// TIA Portal V15.1 export
// export: Created 2024-05-17T05:38:30.0630205Z, ExportSetting WithDefaults, DisplayName Totally Integrated Automation Portal, DisplayVersion V15.1 Update 5, DisplayName TIA Portal Openness, DisplayVersion V15.1 Update 5, DisplayName SINAMICS Startdrive Advanced, DisplayVersion V15.1, DisplayName G130, G150, S120, S150, SINAMICS MV, S210, DisplayVersion V15.1, DisplayName G110M, G120, G120C, G120D, G120P, DisplayVersion V15.1, DisplayName STEP 7 Professional, DisplayVersion V15.1 Update 5, DisplayName STEP 7 Safety, DisplayVersion V15.1, DisplayName WinCC Professional, DisplayVersion V15.1 Update 5, DisplayName SIMATIC Visualization Architect, DisplayVersion V15.1
FUNCTION_BLOCK "LComAlarm"   // FB2105, FBD
TITLE = LComAlarm
{ S7_Optimized_Access := 'FALSE' }
AUTHOR : VCC
FAMILY : Communic
VERSION : 0.1
// =============================================================================
// This module Handles All Alarm Report To MES/VD
// =============================================================================
// stored: AutoNumber false, IsIECCheckEnabled false, SetENOAutomatically False, UDAEnableTagReadback false
   VAR_INPUT
      C_VDCommRecvDB { ExternalAccessible := 'False'; ExternalVisible := 'False'; ExternalWritable := 'False'} : DB_ANY;   // VD communication system receive DB; Not to be used by application / VD communication system receive DB; Not to be used by Application
      C_VDCommSendDB { ExternalAccessible := 'False'; ExternalVisible := 'False'; ExternalWritable := 'False'} : DB_ANY;   // VD communication system send DB; Not to be used by application / VD communication system send DB; Not to be used by Application
      C_LocalRecvDB { ExternalAccessible := 'False'; ExternalVisible := 'False'; ExternalWritable := 'False'} : DB_ANY;   // Local DB to store received data; to used by application / Local DB For Recv Data Used By The Application
      C_LocalSendDB { ExternalAccessible := 'False'; ExternalVisible := 'False'; ExternalWritable := 'False'} : DB_ANY;   // Local DB for send data; to be used by application / Local DB For Send Data Used By The Application
      C_GenAlarmDB { ExternalAccessible := 'False'; ExternalVisible := 'False'; ExternalWritable := 'False'} : DB_ANY;   // Alarm DB
      C_AlarmDBMZ1 { ExternalAccessible := 'False'; ExternalVisible := 'False'; ExternalWritable := 'False'} : DB_ANY;   // Alarm DB
      C_AlarmDBMZ2 { ExternalAccessible := 'False'; ExternalVisible := 'False'; ExternalWritable := 'False'} : DB_ANY;   // Alarm DB
      C_AlarmDBMZ3 { ExternalAccessible := 'False'; ExternalVisible := 'False'; ExternalWritable := 'False'} : DB_ANY;   // Alarm DB
      C_AlarmDBMZ4 { ExternalAccessible := 'False'; ExternalVisible := 'False'; ExternalWritable := 'False'} : DB_ANY;   // Alarm DB
      C_AlarmDBMZ5 { ExternalAccessible := 'False'; ExternalVisible := 'False'; ExternalWritable := 'False'} : DB_ANY;   // Alarm DB
      C_AlarmDBMZ6 { ExternalAccessible := 'False'; ExternalVisible := 'False'; ExternalWritable := 'False'} : DB_ANY;   // Alarm DB
      C_AlarmDBMZ7 { ExternalAccessible := 'False'; ExternalVisible := 'False'; ExternalWritable := 'False'} : DB_ANY;   // Alarm DB
      C_AlarmDBMZ8 { ExternalAccessible := 'False'; ExternalVisible := 'False'; ExternalWritable := 'False'} : DB_ANY;   // Alarm DB
      C_AlarmDBMZ9 { ExternalAccessible := 'False'; ExternalVisible := 'False'; ExternalWritable := 'False'} : DB_ANY;   // Alarm DB
      C_AlarmDBMZ10 { ExternalAccessible := 'False'; ExternalVisible := 'False'; ExternalWritable := 'False'} : DB_ANY;   // Alarm DB
      C_AlarmDBMZ11 { ExternalAccessible := 'False'; ExternalVisible := 'False'; ExternalWritable := 'False'} : DB_ANY;   // Alarm DB
      C_AlarmDBMZ12 { ExternalAccessible := 'False'; ExternalVisible := 'False'; ExternalWritable := 'False'} : DB_ANY;   // Alarm DB
      C_AlarmDBMZ13 { ExternalAccessible := 'False'; ExternalVisible := 'False'; ExternalWritable := 'False'} : DB_ANY;   // Alarm DB
      C_AlarmDBMZ14 { ExternalAccessible := 'False'; ExternalVisible := 'False'; ExternalWritable := 'False'} : DB_ANY;   // Alarm DB
      C_GenAlarmCompare { ExternalAccessible := 'False'; ExternalVisible := 'False'; ExternalWritable := 'False'} : DB_ANY;   // Alarm DB
      C_AlarmCompareDBMZ1 { ExternalAccessible := 'False'; ExternalVisible := 'False'; ExternalWritable := 'False'} : DB_ANY;   // Alarm DB
      C_AlarmCompareDBMZ2 { ExternalAccessible := 'False'; ExternalVisible := 'False'; ExternalWritable := 'False'} : DB_ANY;   // Alarm DB
      C_AlarmCompareDBMZ3 { ExternalAccessible := 'False'; ExternalVisible := 'False'; ExternalWritable := 'False'} : DB_ANY;   // Alarm DB
      C_AlarmCompareDBMZ4 { ExternalAccessible := 'False'; ExternalVisible := 'False'; ExternalWritable := 'False'} : DB_ANY;   // Alarm DB
      C_AlarmCompareDBMZ5 { ExternalAccessible := 'False'; ExternalVisible := 'False'; ExternalWritable := 'False'} : DB_ANY;   // Alarm DB
      C_AlarmCompareDBMZ6 { ExternalAccessible := 'False'; ExternalVisible := 'False'; ExternalWritable := 'False'} : DB_ANY;   // Alarm DB
      C_AlarmCompareDBMZ7 { ExternalAccessible := 'False'; ExternalVisible := 'False'; ExternalWritable := 'False'} : DB_ANY;   // Alarm DB
      C_AlarmCompareDBMZ8 { ExternalAccessible := 'False'; ExternalVisible := 'False'; ExternalWritable := 'False'} : DB_ANY;   // Alarm DB
      C_AlarmCompareDBMZ9 { ExternalAccessible := 'False'; ExternalVisible := 'False'; ExternalWritable := 'False'} : DB_ANY;   // Alarm DB
      C_AlarmCompareDBMZ10 { ExternalAccessible := 'False'; ExternalVisible := 'False'; ExternalWritable := 'False'} : DB_ANY;   // Alarm DB
      C_AlarmCompareDBMZ11 { ExternalAccessible := 'False'; ExternalVisible := 'False'; ExternalWritable := 'False'} : DB_ANY;   // Alarm DB
      C_AlarmCompareDBMZ12 { ExternalAccessible := 'False'; ExternalVisible := 'False'; ExternalWritable := 'False'} : DB_ANY;   // Alarm DB
      C_AlarmCompareDBMZ13 { ExternalAccessible := 'False'; ExternalVisible := 'False'; ExternalWritable := 'False'} : DB_ANY;   // Alarm DB
      C_AlarmCompareDBMZ14 { ExternalAccessible := 'False'; ExternalVisible := 'False'; ExternalWritable := 'False'} : DB_ANY;   // Alarm DB
      C_SubSystem { ExternalAccessible := 'False'; ExternalVisible := 'False'; ExternalWritable := 'False'} : Int;   // Number to identify the subsystem / Identify Subsystem
      C_SendDelay { ExternalAccessible := 'False'; ExternalVisible := 'False'; ExternalWritable := 'False'} : DInt;   // Send Alarm Delay
      C_NbrOfModeZone { ExternalAccessible := 'False'; ExternalVisible := 'False'; ExternalWritable := 'False'} : Int;   // Nbr Of ModeZones
      C_Filter { ExternalAccessible := 'False'; ExternalVisible := 'False'; ExternalWritable := 'False'} : Time := T#500ms;   // Filter
   END_VAR
   VAR_IN_OUT
      IO_VD : "VDComm";   // VD Comm
      IO_AlarmDB : "AlarmDB";   // Alarm
   END_VAR
   VAR
      _LVDComSubSystem { ExternalAccessible := 'False'; ExternalVisible := 'False'; ExternalWritable := 'False'; S7_SetPoint := 'True'} : "LVDComSubSystemS7-1500";   // VD Sub System Alarm
   END_VAR
   VAR DB_SPECIFIC
      ReqSendToVDAlarm { ExternalAccessible := 'False'; ExternalVisible := 'False'; ExternalWritable := 'False'} : Array[1..32] of Bool;   // Req VD
      SendAlarm { ExternalAccessible := 'False'; ExternalVisible := 'False'; ExternalWritable := 'False'} : Array[1..64] of Bool;   // Req Send Alarm
      SendAlarmDone { ExternalAccessible := 'False'; ExternalVisible := 'False'; ExternalWritable := 'False'} : Array[1..64] of Bool;   // Change Of State
      ActiveRequest { ExternalAccessible := 'False'; ExternalVisible := 'False'; ExternalWritable := 'False'} : DWord;   // No Requests Active
      OkToRequest { ExternalAccessible := 'False'; ExternalVisible := 'False'; ExternalWritable := 'False'} : Bool;   // Ok To Request New Alarm To VD
      SendDoneVD { ExternalAccessible := 'False'; ExternalVisible := 'False'; ExternalWritable := 'False'} : Bool;   // Request Is Finished
      SendToVD { ExternalAccessible := 'False'; ExternalVisible := 'False'; ExternalWritable := 'False'} : Bool;   // Send To VD
      InitUDT { ExternalAccessible := 'False'; ExternalVisible := 'False'; ExternalWritable := 'False'} : Bool;   // Init
      DelaySend { ExternalAccessible := 'False'; ExternalVisible := 'False'; ExternalWritable := 'False'} : Bool;   // Delay Send To VD
      InitSend { ExternalAccessible := 'False'; ExternalVisible := 'False'; ExternalWritable := 'False'} : Bool;   // Init Send
      ResetSendDone { ExternalAccessible := 'False'; ExternalVisible := 'False'; ExternalWritable := 'False'} : Bool;   // Reset Send Done
      ResetAllRequest { ExternalAccessible := 'False'; ExternalVisible := 'False'; ExternalWritable := 'False'} : Bool;   // Reset All Send Requests
      Edge { ExternalAccessible := 'False'; ExternalVisible := 'False'; ExternalWritable := 'False'} : Array[1..64] of Bool;   // Array
      SendDBNbr { ExternalAccessible := 'False'; ExternalVisible := 'False'; ExternalWritable := 'False'} : Int;   // Pointer
      SendDBBufNbr { ExternalAccessible := 'False'; ExternalVisible := 'False'; ExternalWritable := 'False'} : Int;   // Pointer
      AlarmPointer { ExternalAccessible := 'False'; ExternalVisible := 'False'; ExternalWritable := 'False'} : Word;   // Pointer
      AlarmLength { ExternalAccessible := 'False'; ExternalVisible := 'False'; ExternalWritable := 'False'} : Word;   // Pointer
      SendLength { ExternalAccessible := 'False'; ExternalVisible := 'False'; ExternalWritable := 'False'} : Word;   // Pointer
      SendDoneArr { ExternalAccessible := 'False'; ExternalVisible := 'False'; ExternalWritable := 'False'} : Array[0..1] of DWord;   // Array Send Done
   END_VAR
   VAR
      _DelaySend { ExternalAccessible := 'False'; ExternalVisible := 'False'; ExternalWritable := 'False'; S7_SetPoint := 'True'} : "LTimer";   // FB
      _LMDBToDBGen { ExternalAccessible := 'False'; ExternalVisible := 'False'; ExternalWritable := 'False'; S7_SetPoint := 'True'} : "LMDBToDB";   // FB
      _LMDBToDBMZ1 { ExternalAccessible := 'False'; ExternalVisible := 'False'; ExternalWritable := 'False'; S7_SetPoint := 'True'} : "LMDBToDB";   // FB
      _LMDBToDBMZ2 { ExternalAccessible := 'False'; ExternalVisible := 'False'; ExternalWritable := 'False'; S7_SetPoint := 'True'} : "LMDBToDB";   // FB
      _LMDBToDBMZ3 { ExternalAccessible := 'False'; ExternalVisible := 'False'; ExternalWritable := 'False'; S7_SetPoint := 'True'} : "LMDBToDB";   // FB
      _LMDBToDBMZ4 { ExternalAccessible := 'False'; ExternalVisible := 'False'; ExternalWritable := 'False'; S7_SetPoint := 'True'} : "LMDBToDB";   // FB
      _LMDBToDBMZ5 { ExternalAccessible := 'False'; ExternalVisible := 'False'; ExternalWritable := 'False'; S7_SetPoint := 'True'} : "LMDBToDB";   // FB
      _LMDBToDBMZ6 { ExternalAccessible := 'False'; ExternalVisible := 'False'; ExternalWritable := 'False'; S7_SetPoint := 'True'} : "LMDBToDB";   // FB
      _LMDBToDBMZ7 { ExternalAccessible := 'False'; ExternalVisible := 'False'; ExternalWritable := 'False'; S7_SetPoint := 'True'} : "LMDBToDB";   // FB
      _LMDBToDBMZ8 { ExternalAccessible := 'False'; ExternalVisible := 'False'; ExternalWritable := 'False'; S7_SetPoint := 'True'} : "LMDBToDB";   // FB
      _LMDBToDBMZ9 { ExternalAccessible := 'False'; ExternalVisible := 'False'; ExternalWritable := 'False'; S7_SetPoint := 'True'} : "LMDBToDB";   // FB
      _LMDBToDBMZ10 { ExternalAccessible := 'False'; ExternalVisible := 'False'; ExternalWritable := 'False'; S7_SetPoint := 'True'} : "LMDBToDB";   // FB
      _LMDBToDBMZ11 { ExternalAccessible := 'False'; ExternalVisible := 'False'; ExternalWritable := 'False'; S7_SetPoint := 'True'} : "LMDBToDB";   // FB
      _LMDBToDBMZ12 { ExternalAccessible := 'False'; ExternalVisible := 'False'; ExternalWritable := 'False'; S7_SetPoint := 'True'} : "LMDBToDB";   // FB
      _LMDBToDBMZ13 { ExternalAccessible := 'False'; ExternalVisible := 'False'; ExternalWritable := 'False'; S7_SetPoint := 'True'} : "LMDBToDB";   // FB
      _LMDBToDBMZ14 { ExternalAccessible := 'False'; ExternalVisible := 'False'; ExternalWritable := 'False'; S7_SetPoint := 'True'} : "LMDBToDB";   // FB
      _LDBCheckGen { ExternalAccessible := 'False'; ExternalVisible := 'False'; ExternalWritable := 'False'; S7_SetPoint := 'True'} : "LDBCheck";   // FB
      _LDBCheckMZ1 { ExternalAccessible := 'False'; ExternalVisible := 'False'; ExternalWritable := 'False'; S7_SetPoint := 'True'} : "LDBCheck";   // FB
      _LDBCheckMZ2 { ExternalAccessible := 'False'; ExternalVisible := 'False'; ExternalWritable := 'False'; S7_SetPoint := 'True'} : "LDBCheck";   // FB
      _LDBCheckMZ3 { ExternalAccessible := 'False'; ExternalVisible := 'False'; ExternalWritable := 'False'; S7_SetPoint := 'True'} : "LDBCheck";   // FB
      _LDBCheckMZ4 { ExternalAccessible := 'False'; ExternalVisible := 'False'; ExternalWritable := 'False'; S7_SetPoint := 'True'} : "LDBCheck";   // FB
      _LDBCheckMZ5 { ExternalAccessible := 'False'; ExternalVisible := 'False'; ExternalWritable := 'False'; S7_SetPoint := 'True'} : "LDBCheck";   // FB
      _LDBCheckMZ6 { ExternalAccessible := 'False'; ExternalVisible := 'False'; ExternalWritable := 'False'; S7_SetPoint := 'True'} : "LDBCheck";   // FB
      _LDBCheckMZ7 { ExternalAccessible := 'False'; ExternalVisible := 'False'; ExternalWritable := 'False'; S7_SetPoint := 'True'} : "LDBCheck";   // FB
      _LDBCheckMZ8 { ExternalAccessible := 'False'; ExternalVisible := 'False'; ExternalWritable := 'False'; S7_SetPoint := 'True'} : "LDBCheck";   // FB
      _LDBCheckMZ9 { ExternalAccessible := 'False'; ExternalVisible := 'False'; ExternalWritable := 'False'; S7_SetPoint := 'True'} : "LDBCheck";   // FB
      _LDBCheckMZ10 { ExternalAccessible := 'False'; ExternalVisible := 'False'; ExternalWritable := 'False'; S7_SetPoint := 'True'} : "LDBCheck";   // FB
      _LDBCheckMZ11 { ExternalAccessible := 'False'; ExternalVisible := 'False'; ExternalWritable := 'False'; S7_SetPoint := 'True'} : "LDBCheck";   // FB
      _LDBCheckMZ12 { ExternalAccessible := 'False'; ExternalVisible := 'False'; ExternalWritable := 'False'; S7_SetPoint := 'True'} : "LDBCheck";   // FB
      _LDBCheckMZ13 { ExternalAccessible := 'False'; ExternalVisible := 'False'; ExternalWritable := 'False'; S7_SetPoint := 'True'} : "LDBCheck";   // FB
      _LDBCheckMZ14 { ExternalAccessible := 'False'; ExternalVisible := 'False'; ExternalWritable := 'False'; S7_SetPoint := 'True'} : "LDBCheck";   // FB
   END_VAR
   VAR DB_SPECIFIC
      _SendDoneReset { ExternalAccessible := 'False'; ExternalVisible := 'False'; ExternalWritable := 'False'; S7_SetPoint := 'True'} : TON_TIME;   // FB
      Filter { ExternalAccessible := 'False'; ExternalVisible := 'False'; ExternalWritable := 'False'} : Array[1..16] of Bool;   // Array
      _FilterGen { ExternalAccessible := 'False'; ExternalVisible := 'False'; ExternalWritable := 'False'; S7_SetPoint := 'True'} : TON_TIME;   // FB
      _FilterMZ1 { ExternalAccessible := 'False'; ExternalVisible := 'False'; ExternalWritable := 'False'; S7_SetPoint := 'True'} : TON_TIME;   // FB
      _FilterMZ2 { ExternalAccessible := 'False'; ExternalVisible := 'False'; ExternalWritable := 'False'; S7_SetPoint := 'True'} : TON_TIME;   // FB
      _FilterMZ3 { ExternalAccessible := 'False'; ExternalVisible := 'False'; ExternalWritable := 'False'; S7_SetPoint := 'True'} : TON_TIME;   // FB
      _FilterMZ4 { ExternalAccessible := 'False'; ExternalVisible := 'False'; ExternalWritable := 'False'; S7_SetPoint := 'True'} : TON_TIME;   // FB
      _FilterMZ5 { ExternalAccessible := 'False'; ExternalVisible := 'False'; ExternalWritable := 'False'; S7_SetPoint := 'True'} : TON_TIME;   // FB
      _FilterMZ6 { ExternalAccessible := 'False'; ExternalVisible := 'False'; ExternalWritable := 'False'; S7_SetPoint := 'True'} : TON_TIME;   // FB
      _FilterMZ7 { ExternalAccessible := 'False'; ExternalVisible := 'False'; ExternalWritable := 'False'; S7_SetPoint := 'True'} : TON_TIME;   // FB
      _FilterMZ8 { ExternalAccessible := 'False'; ExternalVisible := 'False'; ExternalWritable := 'False'; S7_SetPoint := 'True'} : TON_TIME;   // FB
      _FilterMZ9 { ExternalAccessible := 'False'; ExternalVisible := 'False'; ExternalWritable := 'False'; S7_SetPoint := 'True'} : TON_TIME;   // FB
      _FilterMZ10 { ExternalAccessible := 'False'; ExternalVisible := 'False'; ExternalWritable := 'False'; S7_SetPoint := 'True'} : TON_TIME;   // FB
      _FilterMZ11 { ExternalAccessible := 'False'; ExternalVisible := 'False'; ExternalWritable := 'False'; S7_SetPoint := 'True'} : TON_TIME;   // FB
      _FilterMZ12 { ExternalAccessible := 'False'; ExternalVisible := 'False'; ExternalWritable := 'False'; S7_SetPoint := 'True'} : TON_TIME;   // FB
      _FilterMZ13 { ExternalAccessible := 'False'; ExternalVisible := 'False'; ExternalWritable := 'False'; S7_SetPoint := 'True'} : TON_TIME;   // FB
      _FilterMZ14 { ExternalAccessible := 'False'; ExternalVisible := 'False'; ExternalWritable := 'False'; S7_SetPoint := 'True'} : TON_TIME;   // FB
      _InitSend { ExternalAccessible := 'False'; ExternalVisible := 'False'; ExternalWritable := 'False'; S7_SetPoint := 'True'} : TON_TIME;   // FB
      GenDBLenghtOk { ExternalAccessible := 'False'; ExternalVisible := 'False'; ExternalWritable := 'False'} : Bool;   // DB Length Ok
      MZ1DBLenghtOk { ExternalAccessible := 'False'; ExternalVisible := 'False'; ExternalWritable := 'False'} : Bool;   // DB Length Ok
      MZ2DBLenghtOk { ExternalAccessible := 'False'; ExternalVisible := 'False'; ExternalWritable := 'False'} : Bool;   // DB Length Ok
      MZ3DBLenghtOk { ExternalAccessible := 'False'; ExternalVisible := 'False'; ExternalWritable := 'False'} : Bool;   // DB Length Ok
      MZ4DBLenghtOk { ExternalAccessible := 'False'; ExternalVisible := 'False'; ExternalWritable := 'False'} : Bool;   // DB Length Ok
      MZ5DBLenghtOk { ExternalAccessible := 'False'; ExternalVisible := 'False'; ExternalWritable := 'False'} : Bool;   // DB Length Ok
      MZ6DBLenghtOk { ExternalAccessible := 'False'; ExternalVisible := 'False'; ExternalWritable := 'False'} : Bool;   // DB Length Ok
      MZ7DBLenghtOk { ExternalAccessible := 'False'; ExternalVisible := 'False'; ExternalWritable := 'False'} : Bool;   // DB Length Ok
      MZ8DBLenghtOk { ExternalAccessible := 'False'; ExternalVisible := 'False'; ExternalWritable := 'False'} : Bool;   // DB Length Ok
      MZ9DBLenghtOk { ExternalAccessible := 'False'; ExternalVisible := 'False'; ExternalWritable := 'False'} : Bool;   // DB Length Ok
      MZ10DBLenghtOk { ExternalAccessible := 'False'; ExternalVisible := 'False'; ExternalWritable := 'False'} : Bool;   // DB Length Ok
      MZ11DBLenghtOk { ExternalAccessible := 'False'; ExternalVisible := 'False'; ExternalWritable := 'False'} : Bool;   // DB Length Ok
      MZ12DBLenghtOk { ExternalAccessible := 'False'; ExternalVisible := 'False'; ExternalWritable := 'False'} : Bool;   // DB Length Ok
      MZ13DBLenghtOk { ExternalAccessible := 'False'; ExternalVisible := 'False'; ExternalWritable := 'False'} : Bool;   // DB Length Ok
      MZ14DBLenghtOk { ExternalAccessible := 'False'; ExternalVisible := 'False'; ExternalWritable := 'False'} : Bool;   // DB Length Ok
      MZ15DBLenghtOk { ExternalAccessible := 'False'; ExternalVisible := 'False'; ExternalWritable := 'False'} : Bool;   // DB Length Ok
      MZ16DBLenghtOk { ExternalAccessible := 'False'; ExternalVisible := 'False'; ExternalWritable := 'False'} : Bool;   // DB Length Ok
      GenDBLength { ExternalAccessible := 'False'; ExternalVisible := 'False'; ExternalWritable := 'False'} : Word;   // DB Header
      GenDBNumber { ExternalAccessible := 'False'; ExternalVisible := 'False'; ExternalWritable := 'False'} : Word;   // DB Header
      MZ1DBLength { ExternalAccessible := 'False'; ExternalVisible := 'False'; ExternalWritable := 'False'} : Word;   // DB Header
      MZ1DBNumber { ExternalAccessible := 'False'; ExternalVisible := 'False'; ExternalWritable := 'False'} : Word;   // DB Header
      MZ2DBLength { ExternalAccessible := 'False'; ExternalVisible := 'False'; ExternalWritable := 'False'} : Word;   // DB Header
      MZ2DBNumber { ExternalAccessible := 'False'; ExternalVisible := 'False'; ExternalWritable := 'False'} : Word;   // DB Header
      MZ3DBLength { ExternalAccessible := 'False'; ExternalVisible := 'False'; ExternalWritable := 'False'} : Word;   // DB Header
      MZ3DBNumber { ExternalAccessible := 'False'; ExternalVisible := 'False'; ExternalWritable := 'False'} : Word;   // DB Header
      MZ4DBLength { ExternalAccessible := 'False'; ExternalVisible := 'False'; ExternalWritable := 'False'} : Word;   // DB Header
      MZ4DBNumber { ExternalAccessible := 'False'; ExternalVisible := 'False'; ExternalWritable := 'False'} : Word;   // DB Header
      MZ5DBLength { ExternalAccessible := 'False'; ExternalVisible := 'False'; ExternalWritable := 'False'} : Word;   // DB Header
      MZ5DBNumber { ExternalAccessible := 'False'; ExternalVisible := 'False'; ExternalWritable := 'False'} : Word;   // DB Header
      MZ6DBLength { ExternalAccessible := 'False'; ExternalVisible := 'False'; ExternalWritable := 'False'} : Word;   // DB Header
      MZ6DBNumber { ExternalAccessible := 'False'; ExternalVisible := 'False'; ExternalWritable := 'False'} : Word;   // DB Header
      MZ7DBLength { ExternalAccessible := 'False'; ExternalVisible := 'False'; ExternalWritable := 'False'} : Word;   // DB Header
      MZ7DBNumber { ExternalAccessible := 'False'; ExternalVisible := 'False'; ExternalWritable := 'False'} : Word;   // DB Header
      MZ8DBLength { ExternalAccessible := 'False'; ExternalVisible := 'False'; ExternalWritable := 'False'} : Word;   // DB Header
      MZ8DBNumber { ExternalAccessible := 'False'; ExternalVisible := 'False'; ExternalWritable := 'False'} : Word;   // DB Header
      MZ9DBLength { ExternalAccessible := 'False'; ExternalVisible := 'False'; ExternalWritable := 'False'} : Word;   // DB Header
      MZ9DBNumber { ExternalAccessible := 'False'; ExternalVisible := 'False'; ExternalWritable := 'False'} : Word;   // DB Header
      MZ10DBLength { ExternalAccessible := 'False'; ExternalVisible := 'False'; ExternalWritable := 'False'} : Word;   // DB Header
      MZ10DBNumber { ExternalAccessible := 'False'; ExternalVisible := 'False'; ExternalWritable := 'False'} : Word;   // DB Header
      MZ11DBLength { ExternalAccessible := 'False'; ExternalVisible := 'False'; ExternalWritable := 'False'} : Word;   // DB Header
      MZ11DBNumber { ExternalAccessible := 'False'; ExternalVisible := 'False'; ExternalWritable := 'False'} : Word;   // DB Header
      MZ12DBLength { ExternalAccessible := 'False'; ExternalVisible := 'False'; ExternalWritable := 'False'} : Word;   // DB Header
      MZ12DBNumber { ExternalAccessible := 'False'; ExternalVisible := 'False'; ExternalWritable := 'False'} : Word;   // DB Header
      MZ13DBLength { ExternalAccessible := 'False'; ExternalVisible := 'False'; ExternalWritable := 'False'} : Word;   // DB Header
      MZ13DBNumber { ExternalAccessible := 'False'; ExternalVisible := 'False'; ExternalWritable := 'False'} : Word;   // DB Header
      MZ14DBLength { ExternalAccessible := 'False'; ExternalVisible := 'False'; ExternalWritable := 'False'} : Word;   // DB Header
      MZ14DBNumber { ExternalAccessible := 'False'; ExternalVisible := 'False'; ExternalWritable := 'False'} : Word;   // DB Header
      PLCAlarms { ExternalAccessible := 'False'; ExternalVisible := 'False'; ExternalWritable := 'False'; S7_SetPoint := 'True'} : "PLCAlarms";   // Alarm Handling
   END_VAR
   VAR_TEMP
      BPtr : Any;   // Temp
      SPtr : Any;   // Temp
      Pointer : Word;   // Temp
      F : Word;
      GenDBLenghtCompare : Word;   // Temp
      MZ1DBLenghtCompare : Word;   // Temp
      MZ2DBLenghtCompare : Word;   // Temp
      MZ3DBLenghtCompare : Word;   // Temp
      MZ4DBLenghtCompare : Word;   // Temp
      MZ5DBLenghtCompare : Word;   // Temp
      MZ6DBLenghtCompare : Word;   // Temp
      MZ7DBLenghtCompare : Word;   // Temp
      MZ8DBLenghtCompare : Word;   // Temp
      MZ9DBLenghtCompare : Word;   // Temp
      MZ10DBLenghtCompare : Word;   // Temp
      MZ11DBLenghtCompare : Word;   // Temp
      MZ12DBLenghtCompare : Word;   // Temp
      MZ13DBLenghtCompare : Word;   // Temp
      MZ14DBLenghtCompare : Word;   // Temp
      GenOk : Bool;   // Temp
      MZ1Ok : Bool;   // Temp
      MZ2Ok : Bool;   // Temp
      MZ3Ok : Bool;   // Temp
      MZ4Ok : Bool;   // Temp
      MZ5Ok : Bool;   // Temp
      MZ6Ok : Bool;   // Temp
      MZ7Ok : Bool;   // Temp
      MZ8Ok : Bool;   // Temp
      MZ9Ok : Bool;   // Temp
      MZ10Ok : Bool;   // Temp
      MZ11Ok : Bool;   // Temp
      MZ12Ok : Bool;   // Temp
      MZ13Ok : Bool;   // Temp
      MZ14Ok : Bool;   // Temp
   END_VAR
   VAR_TEMP   // added for the SCL form of the ladder/FBD networks
      _w1 : Bool;
   END_VAR
BEGIN

REGION Network 1: **** 3.1 - Communication - Other Systems **** Request Event To VD
   // Request Send To VD
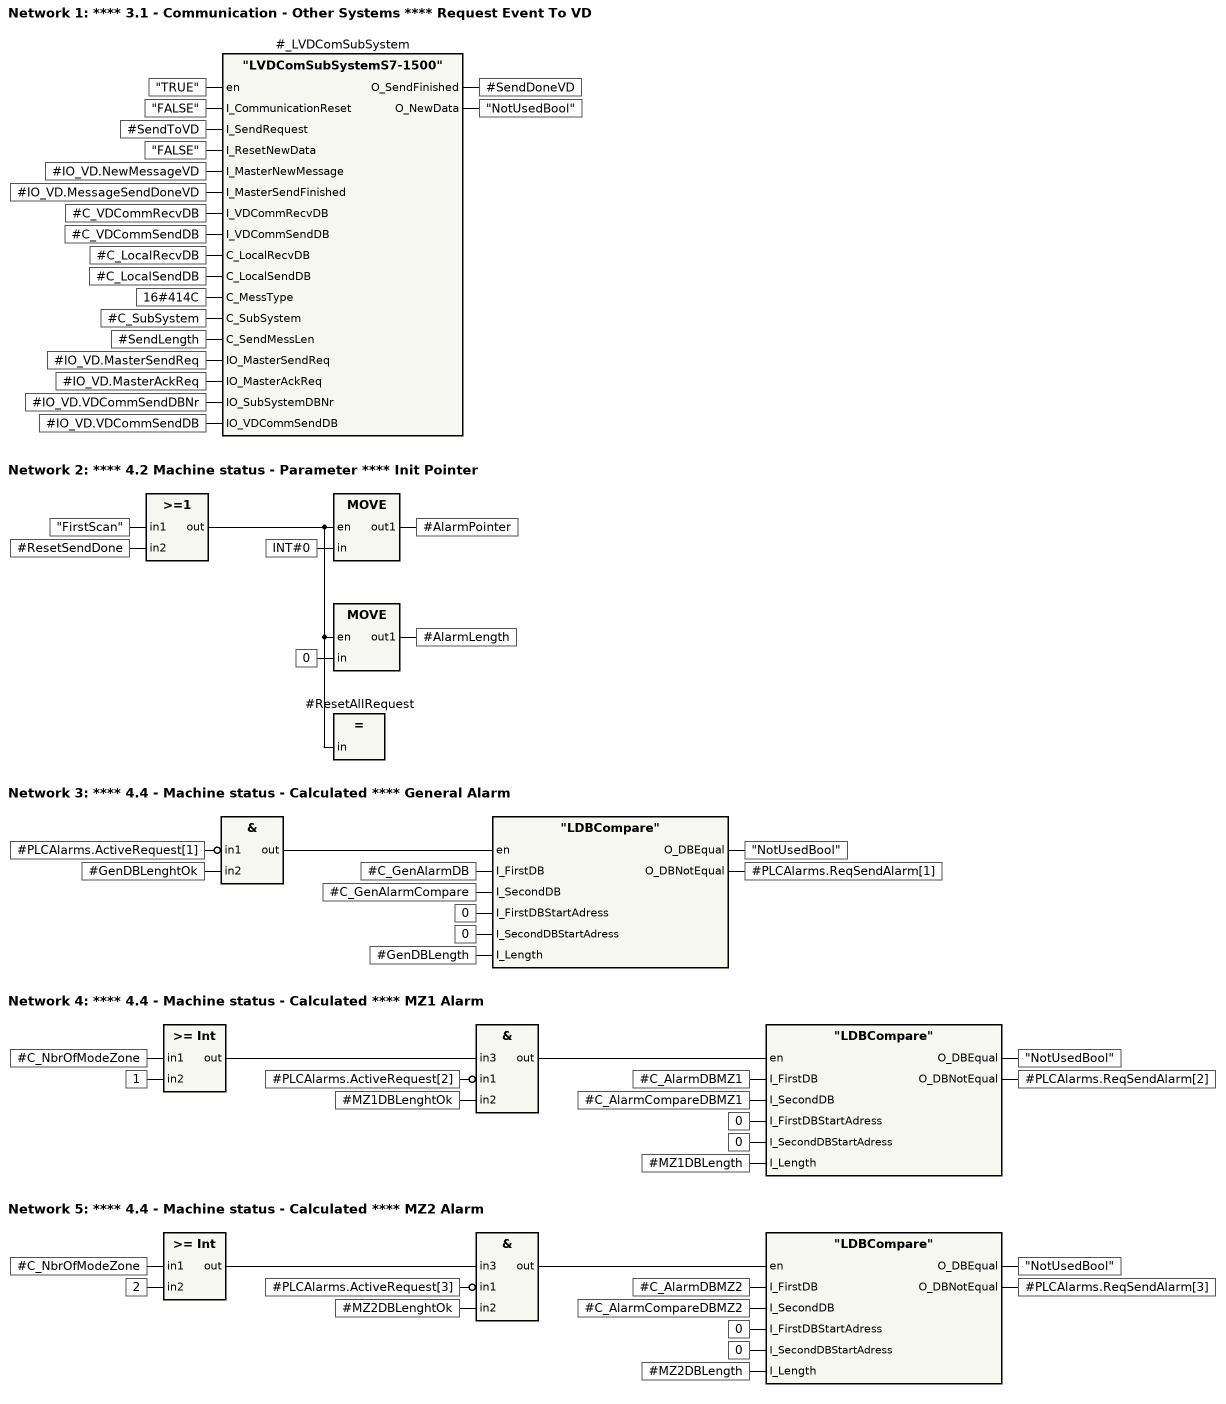
   IF "TRUE" THEN
       #_LVDComSubSystem(I_CommunicationReset := "FALSE",   // "LVDComSubSystemS7-1500"
                         I_SendRequest := #SendToVD,
                         I_ResetNewData := "FALSE",
                         I_MasterNewMessage := #IO_VD.NewMessageVD,
                         I_MasterSendFinished := #IO_VD.MessageSendDoneVD,
                         I_VDCommRecvDB := #C_VDCommRecvDB,
                         I_VDCommSendDB := #C_VDCommSendDB,
                         C_LocalRecvDB := #C_LocalRecvDB,
                         C_LocalSendDB := #C_LocalSendDB,
                         C_MessType := 16#414C,
                         C_SubSystem := #C_SubSystem,
                         C_SendMessLen := #SendLength,
                         IO_MasterSendReq := #IO_VD.MasterSendReq,
                         IO_MasterAckReq := #IO_VD.MasterAckReq,
                         IO_SubSystemDBNr := #IO_VD.VDCommSendDBNr,
                         IO_VDCommSendDB := #IO_VD.VDCommSendDB,
                         O_SendFinished => #SendDoneVD,
                         O_NewData => "NotUsedBool");
   END_IF;
END_REGION

REGION Network 2: **** 4.2 Machine status - Parameter **** Init Pointer
   // Init Pointer
   #_w1 := "FirstScan" OR #ResetSendDone;
   IF #_w1 THEN
       #AlarmPointer := INT#0;
       #AlarmLength := 0;
   END_IF;
   #ResetAllRequest := #_w1;
END_REGION

REGION Network 3: **** 4.4 - Machine status - Calculated **** General Alarm
   // Check If There Is New Alarms
   IF NOT #PLCAlarms.ActiveRequest[1] AND #GenDBLenghtOk THEN
       "LDBCompare"(I_FirstDB := #C_GenAlarmDB,
                    I_SecondDB := #C_GenAlarmCompare,
                    I_FirstDBStartAdress := 0,
                    I_SecondDBStartAdress := 0,
                    I_Length := #GenDBLength,
                    O_DBEqual => "NotUsedBool",
                    O_DBNotEqual => #PLCAlarms.ReqSendAlarm[1]);
   END_IF;
END_REGION

REGION Network 4: **** 4.4 - Machine status - Calculated **** MZ1 Alarm
   // Check If There Is New Alarms
   IF (#C_NbrOfModeZone >= 1) AND NOT #PLCAlarms.ActiveRequest[2] AND #MZ1DBLenghtOk THEN
       "LDBCompare"(I_FirstDB := #C_AlarmDBMZ1,
                    I_SecondDB := #C_AlarmCompareDBMZ1,
                    I_FirstDBStartAdress := 0,
                    I_SecondDBStartAdress := 0,
                    I_Length := #MZ1DBLength,
                    O_DBEqual => "NotUsedBool",
                    O_DBNotEqual => #PLCAlarms.ReqSendAlarm[2]);
   END_IF;
END_REGION

REGION Network 5: **** 4.4 - Machine status - Calculated **** MZ2 Alarm
   // Check If There Is New Alarms
   IF (#C_NbrOfModeZone >= 2) AND NOT #PLCAlarms.ActiveRequest[3] AND #MZ2DBLenghtOk THEN
       "LDBCompare"(I_FirstDB := #C_AlarmDBMZ2,
                    I_SecondDB := #C_AlarmCompareDBMZ2,
                    I_FirstDBStartAdress := 0,
                    I_SecondDBStartAdress := 0,
                    I_Length := #MZ2DBLength,
                    O_DBEqual => "NotUsedBool",
                    O_DBNotEqual => #PLCAlarms.ReqSendAlarm[3]);
   END_IF;
END_REGION

REGION Network 6: **** 4.4 - Machine status - Calculated **** MZ3 Alarm
   // Check If There Is New Alarms
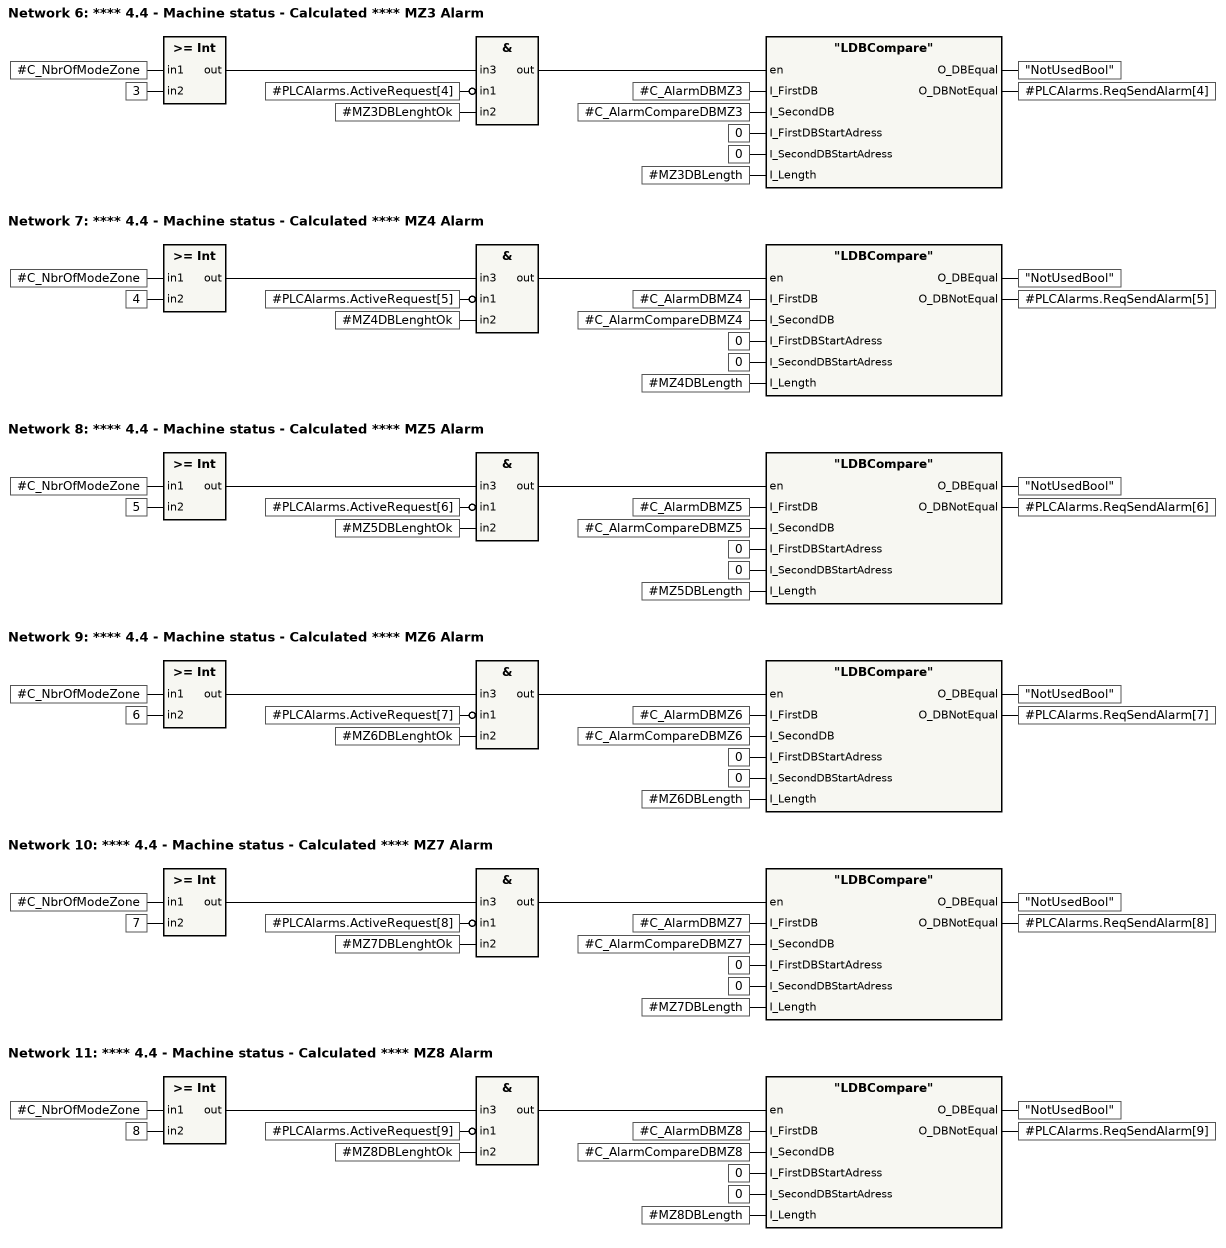
   IF (#C_NbrOfModeZone >= 3) AND NOT #PLCAlarms.ActiveRequest[4] AND #MZ3DBLenghtOk THEN
       "LDBCompare"(I_FirstDB := #C_AlarmDBMZ3,
                    I_SecondDB := #C_AlarmCompareDBMZ3,
                    I_FirstDBStartAdress := 0,
                    I_SecondDBStartAdress := 0,
                    I_Length := #MZ3DBLength,
                    O_DBEqual => "NotUsedBool",
                    O_DBNotEqual => #PLCAlarms.ReqSendAlarm[4]);
   END_IF;
END_REGION

REGION Network 7: **** 4.4 - Machine status - Calculated **** MZ4 Alarm
   // Check If There Is New Alarms
   IF (#C_NbrOfModeZone >= 4) AND NOT #PLCAlarms.ActiveRequest[5] AND #MZ4DBLenghtOk THEN
       "LDBCompare"(I_FirstDB := #C_AlarmDBMZ4,
                    I_SecondDB := #C_AlarmCompareDBMZ4,
                    I_FirstDBStartAdress := 0,
                    I_SecondDBStartAdress := 0,
                    I_Length := #MZ4DBLength,
                    O_DBEqual => "NotUsedBool",
                    O_DBNotEqual => #PLCAlarms.ReqSendAlarm[5]);
   END_IF;
END_REGION

REGION Network 8: **** 4.4 - Machine status - Calculated **** MZ5 Alarm
   // Check If There Is New Alarms
   IF (#C_NbrOfModeZone >= 5) AND NOT #PLCAlarms.ActiveRequest[6] AND #MZ5DBLenghtOk THEN
       "LDBCompare"(I_FirstDB := #C_AlarmDBMZ5,
                    I_SecondDB := #C_AlarmCompareDBMZ5,
                    I_FirstDBStartAdress := 0,
                    I_SecondDBStartAdress := 0,
                    I_Length := #MZ5DBLength,
                    O_DBEqual => "NotUsedBool",
                    O_DBNotEqual => #PLCAlarms.ReqSendAlarm[6]);
   END_IF;
END_REGION

REGION Network 9: **** 4.4 - Machine status - Calculated **** MZ6 Alarm
   // Check If There Is New Alarms
   IF (#C_NbrOfModeZone >= 6) AND NOT #PLCAlarms.ActiveRequest[7] AND #MZ6DBLenghtOk THEN
       "LDBCompare"(I_FirstDB := #C_AlarmDBMZ6,
                    I_SecondDB := #C_AlarmCompareDBMZ6,
                    I_FirstDBStartAdress := 0,
                    I_SecondDBStartAdress := 0,
                    I_Length := #MZ6DBLength,
                    O_DBEqual => "NotUsedBool",
                    O_DBNotEqual => #PLCAlarms.ReqSendAlarm[7]);
   END_IF;
END_REGION

REGION Network 10: **** 4.4 - Machine status - Calculated **** MZ7 Alarm
   // Check If There Is New Alarms
   IF (#C_NbrOfModeZone >= 7) AND NOT #PLCAlarms.ActiveRequest[8] AND #MZ7DBLenghtOk THEN
       "LDBCompare"(I_FirstDB := #C_AlarmDBMZ7,
                    I_SecondDB := #C_AlarmCompareDBMZ7,
                    I_FirstDBStartAdress := 0,
                    I_SecondDBStartAdress := 0,
                    I_Length := #MZ7DBLength,
                    O_DBEqual => "NotUsedBool",
                    O_DBNotEqual => #PLCAlarms.ReqSendAlarm[8]);
   END_IF;
END_REGION

REGION Network 11: **** 4.4 - Machine status - Calculated **** MZ8 Alarm
   // Check If There Is New Alarms
   IF (#C_NbrOfModeZone >= 8) AND NOT #PLCAlarms.ActiveRequest[9] AND #MZ8DBLenghtOk THEN
       "LDBCompare"(I_FirstDB := #C_AlarmDBMZ8,
                    I_SecondDB := #C_AlarmCompareDBMZ8,
                    I_FirstDBStartAdress := 0,
                    I_SecondDBStartAdress := 0,
                    I_Length := #MZ8DBLength,
                    O_DBEqual => "NotUsedBool",
                    O_DBNotEqual => #PLCAlarms.ReqSendAlarm[9]);
   END_IF;
END_REGION

REGION Network 12: **** 4.4 - Machine status - Calculated **** MZ9 Alarm
   // Check If There Is New Alarms
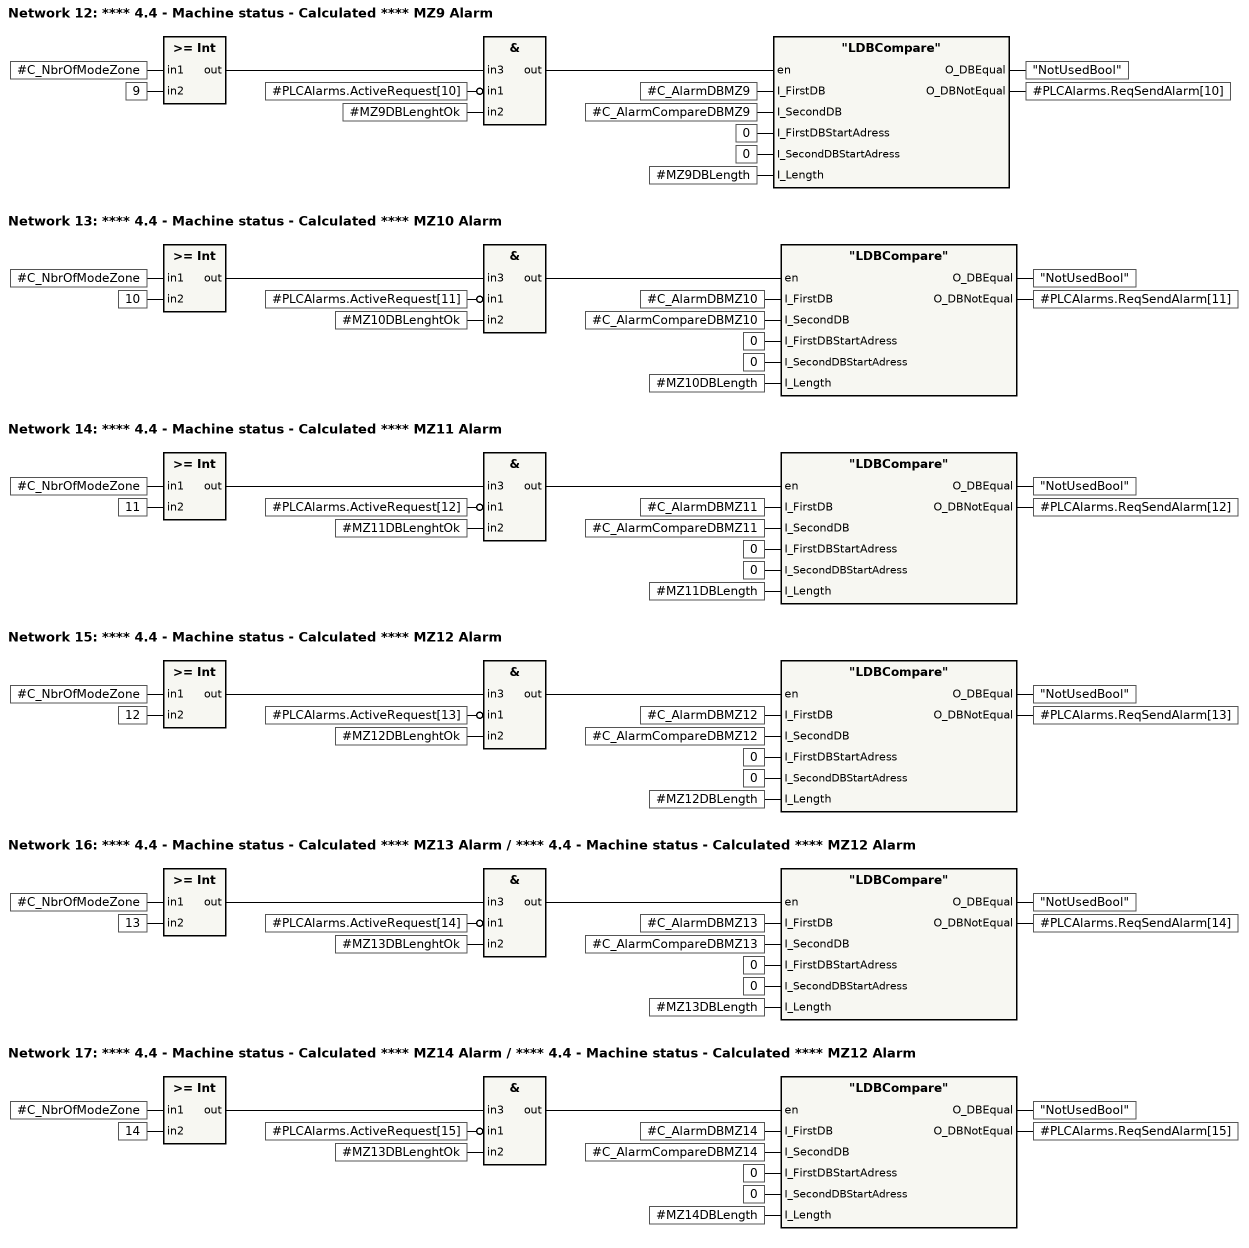
   IF (#C_NbrOfModeZone >= 9) AND NOT #PLCAlarms.ActiveRequest[10] AND #MZ9DBLenghtOk THEN
       "LDBCompare"(I_FirstDB := #C_AlarmDBMZ9,
                    I_SecondDB := #C_AlarmCompareDBMZ9,
                    I_FirstDBStartAdress := 0,
                    I_SecondDBStartAdress := 0,
                    I_Length := #MZ9DBLength,
                    O_DBEqual => "NotUsedBool",
                    O_DBNotEqual => #PLCAlarms.ReqSendAlarm[10]);
   END_IF;
END_REGION

REGION Network 13: **** 4.4 - Machine status - Calculated **** MZ10 Alarm
   // Check If There Is New Alarms
   IF (#C_NbrOfModeZone >= 10) AND NOT #PLCAlarms.ActiveRequest[11] AND #MZ10DBLenghtOk THEN
       "LDBCompare"(I_FirstDB := #C_AlarmDBMZ10,
                    I_SecondDB := #C_AlarmCompareDBMZ10,
                    I_FirstDBStartAdress := 0,
                    I_SecondDBStartAdress := 0,
                    I_Length := #MZ10DBLength,
                    O_DBEqual => "NotUsedBool",
                    O_DBNotEqual => #PLCAlarms.ReqSendAlarm[11]);
   END_IF;
END_REGION

REGION Network 14: **** 4.4 - Machine status - Calculated **** MZ11 Alarm
   // Check If There Is New Alarms
   IF (#C_NbrOfModeZone >= 11) AND NOT #PLCAlarms.ActiveRequest[12] AND #MZ11DBLenghtOk THEN
       "LDBCompare"(I_FirstDB := #C_AlarmDBMZ11,
                    I_SecondDB := #C_AlarmCompareDBMZ11,
                    I_FirstDBStartAdress := 0,
                    I_SecondDBStartAdress := 0,
                    I_Length := #MZ11DBLength,
                    O_DBEqual => "NotUsedBool",
                    O_DBNotEqual => #PLCAlarms.ReqSendAlarm[12]);
   END_IF;
END_REGION

REGION Network 15: **** 4.4 - Machine status - Calculated **** MZ12 Alarm
   // Check If There Is New Alarms
   IF (#C_NbrOfModeZone >= 12) AND NOT #PLCAlarms.ActiveRequest[13] AND #MZ12DBLenghtOk THEN
       "LDBCompare"(I_FirstDB := #C_AlarmDBMZ12,
                    I_SecondDB := #C_AlarmCompareDBMZ12,
                    I_FirstDBStartAdress := 0,
                    I_SecondDBStartAdress := 0,
                    I_Length := #MZ12DBLength,
                    O_DBEqual => "NotUsedBool",
                    O_DBNotEqual => #PLCAlarms.ReqSendAlarm[13]);
   END_IF;
END_REGION

REGION Network 16: **** 4.4 - Machine status - Calculated **** MZ13 Alarm / **** 4.4 - Machine status - Calculated **** MZ12 Alarm
   // Check If There Is New Alarms
   IF (#C_NbrOfModeZone >= 13) AND NOT #PLCAlarms.ActiveRequest[14] AND #MZ13DBLenghtOk THEN
       "LDBCompare"(I_FirstDB := #C_AlarmDBMZ13,
                    I_SecondDB := #C_AlarmCompareDBMZ13,
                    I_FirstDBStartAdress := 0,
                    I_SecondDBStartAdress := 0,
                    I_Length := #MZ13DBLength,
                    O_DBEqual => "NotUsedBool",
                    O_DBNotEqual => #PLCAlarms.ReqSendAlarm[14]);
   END_IF;
END_REGION

REGION Network 17: **** 4.4 - Machine status - Calculated **** MZ14 Alarm / **** 4.4 - Machine status - Calculated **** MZ12 Alarm
   // Check If There Is New Alarms
   IF (#C_NbrOfModeZone >= 14) AND NOT #PLCAlarms.ActiveRequest[15] AND #MZ13DBLenghtOk THEN
       "LDBCompare"(I_FirstDB := #C_AlarmDBMZ14,
                    I_SecondDB := #C_AlarmCompareDBMZ14,
                    I_FirstDBStartAdress := 0,
                    I_SecondDBStartAdress := 0,
                    I_Length := #MZ14DBLength,
                    O_DBEqual => "NotUsedBool",
                    O_DBNotEqual => #PLCAlarms.ReqSendAlarm[15]);
   END_IF;
END_REGION

REGION Network 18: **** 4.4 - Machine status - Calculated **** Erase All Requests
   // Erase All Requests
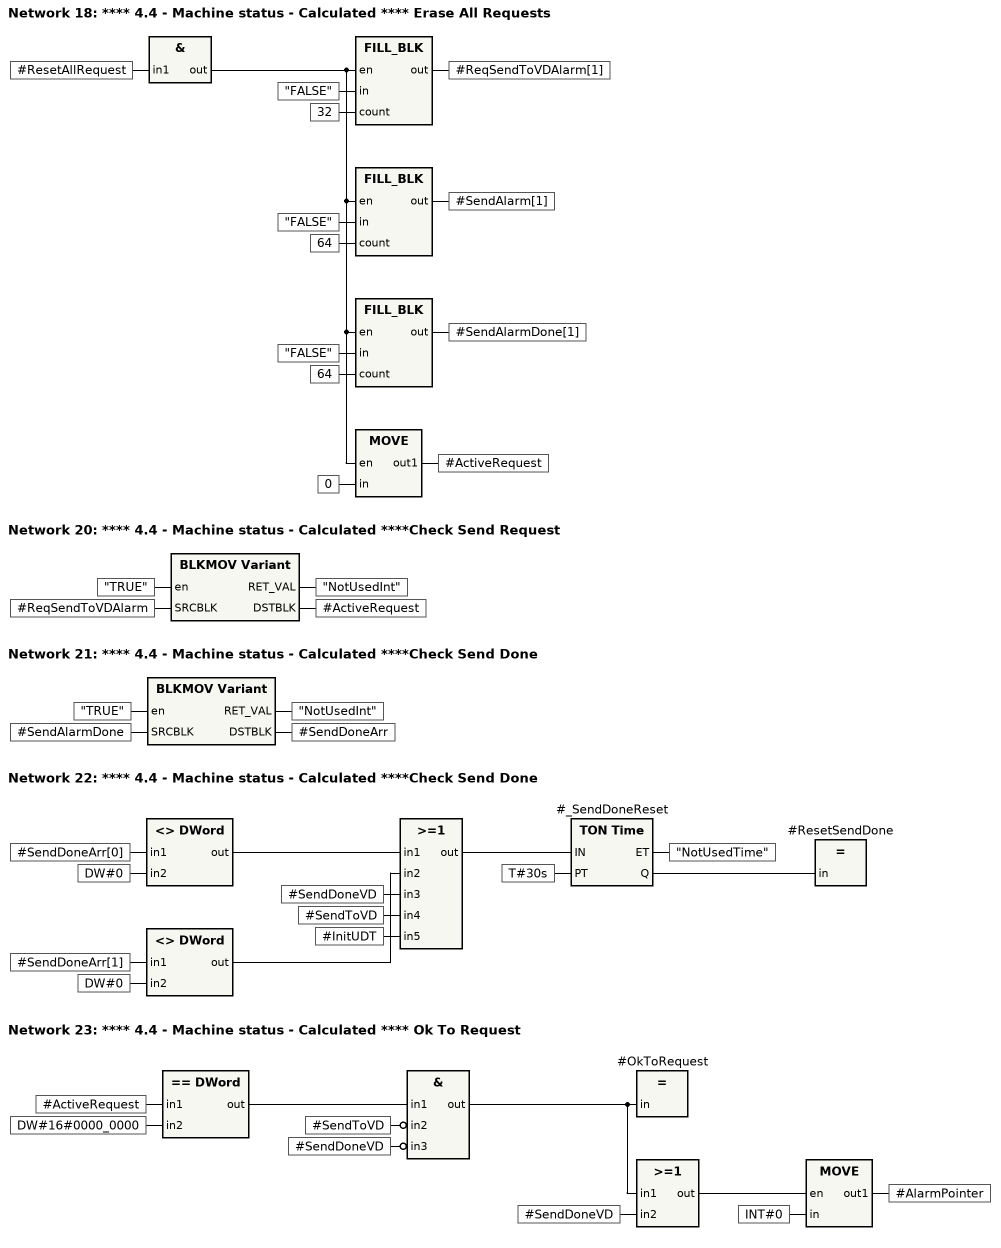
   IF #ResetAllRequest THEN
       FILL_BLK(IN := "FALSE", COUNT := 32, OUT => #ReqSendToVDAlarm[1]);
       FILL_BLK(IN := "FALSE", COUNT := 64, OUT => #SendAlarm[1]);
       FILL_BLK(IN := "FALSE", COUNT := 64, OUT => #SendAlarmDone[1]);
       #ActiveRequest := 0;
   END_IF;
END_REGION

NETWORK
TITLE = **** 4.4 - Machine status - Calculated **** Init UDT
// Init UDT
      A     #ResetAllRequest;
      O     #ResetSendDone;
      JCN   NoInit;
      R     #PLCAlarms.ReqSendAlarm[1];
      R     #PLCAlarms.ReqSendAlarm[2];
      R     #PLCAlarms.ReqSendAlarm[3];
      R     #PLCAlarms.ReqSendAlarm[4];
      R     #PLCAlarms.ReqSendAlarm[5];
      R     #PLCAlarms.ReqSendAlarm[6];
      R     #PLCAlarms.ReqSendAlarm[7];
      R     #PLCAlarms.ReqSendAlarm[8];
      R     #PLCAlarms.ReqSendAlarm[9];
      R     #PLCAlarms.ReqSendAlarm[10];
      R     #PLCAlarms.ReqSendAlarm[11];
      R     #PLCAlarms.ReqSendAlarm[12];
      R     #PLCAlarms.ReqSendAlarm[13];
      R     #PLCAlarms.ReqSendAlarm[14];
      R     #PLCAlarms.ReqSendAlarm[15];
      R     #PLCAlarms.ReqSendAlarm[16];
      R     #PLCAlarms.ReqSendAlarm[17];
      R     #PLCAlarms.ReqSendAlarm[18];
      R     #PLCAlarms.ReqSendAlarm[19];
      R     #PLCAlarms.ReqSendAlarm[20];
      R     #PLCAlarms.ReqSendAlarm[21];
      R     #PLCAlarms.ReqSendAlarm[22];
      R     #PLCAlarms.ReqSendAlarm[23];
      R     #PLCAlarms.ReqSendAlarm[24];
      R     #PLCAlarms.ReqSendAlarm[25];
      R     #PLCAlarms.ReqSendAlarm[26];
      R     #PLCAlarms.ReqSendAlarm[27];
      R     #PLCAlarms.ReqSendAlarm[28];
      R     #PLCAlarms.ReqSendAlarm[29];
      R     #PLCAlarms.ReqSendAlarm[30];
      R     #PLCAlarms.ReqSendAlarm[31];
      R     #PLCAlarms.ReqSendAlarm[32];
      R     #PLCAlarms.ActiveRequest[1];
      R     #PLCAlarms.ActiveRequest[2];
      R     #PLCAlarms.ActiveRequest[3];
      R     #PLCAlarms.ActiveRequest[4];
      R     #PLCAlarms.ActiveRequest[5];
      R     #PLCAlarms.ActiveRequest[6];
      R     #PLCAlarms.ActiveRequest[7];
      R     #PLCAlarms.ActiveRequest[8];
      R     #PLCAlarms.ActiveRequest[9];
      R     #PLCAlarms.ActiveRequest[10];
      R     #PLCAlarms.ActiveRequest[11];
      R     #PLCAlarms.ActiveRequest[12];
      R     #PLCAlarms.ActiveRequest[13];
      R     #PLCAlarms.ActiveRequest[14];
      R     #PLCAlarms.ActiveRequest[15];
      R     #PLCAlarms.ActiveRequest[16];
      R     #PLCAlarms.ActiveRequest[17];
      R     #PLCAlarms.ActiveRequest[18];
      R     #PLCAlarms.ActiveRequest[19];
      R     #PLCAlarms.ActiveRequest[20];
      R     #PLCAlarms.ActiveRequest[21];
      R     #PLCAlarms.ActiveRequest[22];
      R     #PLCAlarms.ActiveRequest[23];
      R     #PLCAlarms.ActiveRequest[24];
      R     #PLCAlarms.ActiveRequest[25];
      R     #PLCAlarms.ActiveRequest[26];
      R     #PLCAlarms.ActiveRequest[27];
      R     #PLCAlarms.ActiveRequest[28];
      R     #PLCAlarms.ActiveRequest[29];
      R     #PLCAlarms.ActiveRequest[30];
      R     #PLCAlarms.ActiveRequest[31];
      R     #PLCAlarms.ActiveRequest[32];

NoInit:NOP   0;

      A     #PLCAlarms.ReqSendAlarm[1];
      O     #PLCAlarms.ReqSendAlarm[2];
      O     #PLCAlarms.ReqSendAlarm[3];
      O     #PLCAlarms.ReqSendAlarm[4];
      O     #PLCAlarms.ReqSendAlarm[5];
      O     #PLCAlarms.ReqSendAlarm[6];
      O     #PLCAlarms.ReqSendAlarm[7];
      O     #PLCAlarms.ReqSendAlarm[8];
      O     #PLCAlarms.ReqSendAlarm[9];
      O     #PLCAlarms.ReqSendAlarm[10];
      O     #PLCAlarms.ReqSendAlarm[11];
      O     #PLCAlarms.ReqSendAlarm[12];
      O     #PLCAlarms.ReqSendAlarm[13];
      O     #PLCAlarms.ReqSendAlarm[14];
      O     #PLCAlarms.ReqSendAlarm[15];
      O     #PLCAlarms.ReqSendAlarm[16];
      O     #PLCAlarms.ReqSendAlarm[17];
      O     #PLCAlarms.ReqSendAlarm[18];
      O     #PLCAlarms.ReqSendAlarm[19];
      O     #PLCAlarms.ReqSendAlarm[20];
      O     #PLCAlarms.ReqSendAlarm[21];
      O     #PLCAlarms.ReqSendAlarm[22];
      O     #PLCAlarms.ReqSendAlarm[23];
      O     #PLCAlarms.ReqSendAlarm[24];
      O     #PLCAlarms.ReqSendAlarm[25];
      O     #PLCAlarms.ReqSendAlarm[26];
      O     #PLCAlarms.ReqSendAlarm[27];
      O     #PLCAlarms.ReqSendAlarm[28];
      O     #PLCAlarms.ReqSendAlarm[29];
      O     #PLCAlarms.ReqSendAlarm[30];
      O     #PLCAlarms.ReqSendAlarm[31];
      O     #PLCAlarms.ReqSendAlarm[32];
      O     #PLCAlarms.ActiveRequest[1];
      O     #PLCAlarms.ActiveRequest[2];
      O     #PLCAlarms.ActiveRequest[3];
      O     #PLCAlarms.ActiveRequest[4];
      O     #PLCAlarms.ActiveRequest[5];
      O     #PLCAlarms.ActiveRequest[6];
      O     #PLCAlarms.ActiveRequest[7];
      O     #PLCAlarms.ActiveRequest[8];
      O     #PLCAlarms.ActiveRequest[9];
      O     #PLCAlarms.ActiveRequest[10];
      O     #PLCAlarms.ActiveRequest[11];
      O     #PLCAlarms.ActiveRequest[12];
      O     #PLCAlarms.ActiveRequest[13];
      O     #PLCAlarms.ActiveRequest[14];
      O     #PLCAlarms.ActiveRequest[15];
      O     #PLCAlarms.ActiveRequest[16];
      O     #PLCAlarms.ActiveRequest[17];
      O     #PLCAlarms.ActiveRequest[18];
      O     #PLCAlarms.ActiveRequest[19];
      O     #PLCAlarms.ActiveRequest[20];
      O     #PLCAlarms.ActiveRequest[21];
      O     #PLCAlarms.ActiveRequest[22];
      O     #PLCAlarms.ActiveRequest[23];
      O     #PLCAlarms.ActiveRequest[24];
      O     #PLCAlarms.ActiveRequest[25];
      O     #PLCAlarms.ActiveRequest[26];
      O     #PLCAlarms.ActiveRequest[27];
      O     #PLCAlarms.ActiveRequest[28];
      O     #PLCAlarms.ActiveRequest[29];
      O     #PLCAlarms.ActiveRequest[30];
      O     #PLCAlarms.ActiveRequest[31];
      O     #PLCAlarms.ActiveRequest[32];
      =     #InitUDT;


REGION Network 20: **** 4.4 - Machine status - Calculated ****Check Send Request
   // Check Send Request
   IF "TRUE" THEN "NotUsedInt" := BLKMOV(SRCBLK := #ReqSendToVDAlarm, DSTBLK => #ActiveRequest); END_IF;
END_REGION

REGION Network 21: **** 4.4 - Machine status - Calculated ****Check Send Done
   // Check Send Done
   IF "TRUE" THEN "NotUsedInt" := BLKMOV(SRCBLK := #SendAlarmDone, DSTBLK => #SendDoneArr); END_IF;
END_REGION

REGION Network 22: **** 4.4 - Machine status - Calculated ****Check Send Done
   // Check Send Done
   #_SendDoneReset(IN := (#SendDoneArr[0] <> DW#0) OR (#SendDoneArr[1] <> DW#0) OR #SendDoneVD OR #SendToVD OR #InitUDT,   // TON
                   PT := T#30s,
                   ET => "NotUsedTime");
   #ResetSendDone := #_SendDoneReset.Q;
END_REGION

REGION Network 23: **** 4.4 - Machine status - Calculated **** Ok To Request
   // Ok To Request
   #OkToRequest := (#ActiveRequest = DW#16#0000_0000) AND NOT #SendToVD AND NOT #SendDoneVD;
   IF #OkToRequest OR #SendDoneVD THEN #AlarmPointer := INT#0; END_IF;
END_REGION

REGION Network 24: **** 4.4 - Machine status - Calculated **** Delay Send To VD
   // Delay Send To VD
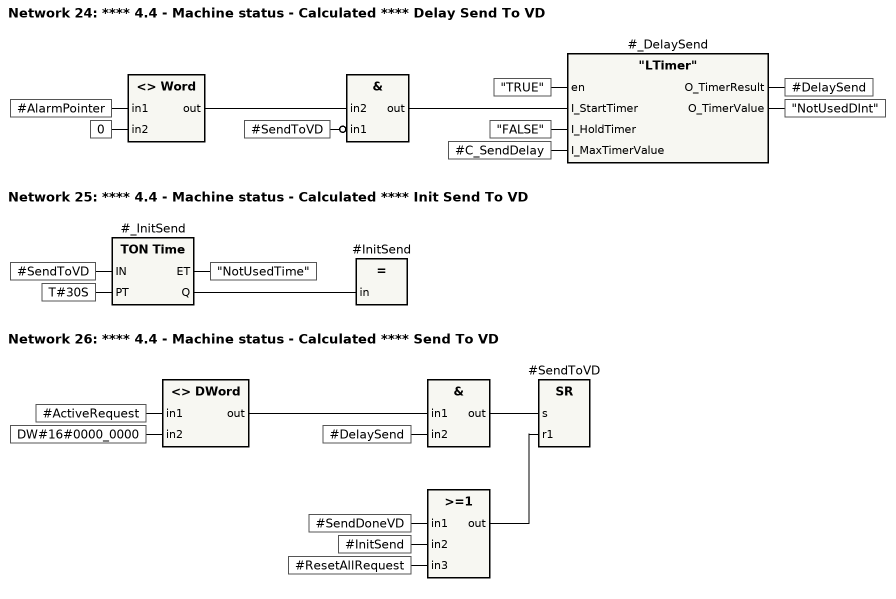
   IF "TRUE" THEN
       #_DelaySend(I_StartTimer := (#AlarmPointer <> 0) AND NOT #SendToVD,   // "LTimer"
                   I_HoldTimer := "FALSE",
                   I_MaxTimerValue := #C_SendDelay,
                   O_TimerResult => #DelaySend,
                   O_TimerValue => "NotUsedDInt");
   END_IF;
END_REGION

REGION Network 25: **** 4.4 - Machine status - Calculated **** Init Send To VD
   // Init Send To VD
   #_InitSend(IN := #SendToVD, PT := T#30S, ET => "NotUsedTime");   // TON
   #InitSend := #_InitSend.Q;
END_REGION

REGION Network 26: **** 4.4 - Machine status - Calculated **** Send To VD
   // Send To VD
   IF (#ActiveRequest <> DW#16#0000_0000) AND #DelaySend THEN
       #SendToVD := TRUE;   // SR flip-flop
   END_IF;
   IF #SendDoneVD OR #InitSend OR #ResetAllRequest THEN #SendToVD := FALSE; END_IF;
END_REGION

NETWORK
TITLE = **** 4.4 - Machine status - Calculated **** Header Send
// Header
// Configure Header For Send Data Alarm, APA// S7-1500 Preparations
      OPN   #C_LocalSendDB;
      L     DBNO;
      T     #SendDBBufNbr;
//    L     #AlarmPointer
//      T     #Pointer
//   OPN DB [ #Pointer]

//      T     #SendDBNbr
//    L DBLG
//  T     #AlarmLength
//
//    NOP 0
      L     #AlarmPointer;
      L     0;
      <>I;
      JCN   NozHeaD;
      L     #AlarmLength;
      +     10;
      T     #SendLength;

      LAR1  P##BPtr;
      L     16#1002;
      T     LW [AR1, P#0.0];
      L     #AlarmLength;
      T     LW [AR1, P#2.0];
      L     #AlarmPointer;
      T     LW [AR1, P#4.0];
      L     0;
      SLD   3;
      OD    16#8400_0000;
      T     LD [AR1, P#6.0];


      LAR1  P##SPtr;
      L     16#1002;
      T     LW [AR1, P#0.0];
      L     #AlarmLength;
      T     LW [AR1, P#2.0];
      L     #SendDBBufNbr;
      T     LW [AR1, P#4.0];
      L     10;
      SLD   3;
      OD    16#8400_0000;
      T     LD [AR1, P#6.0];
      CALL  BLKMOV
      ( SRCBLK  := #BPtr,
        RET_VAL := "NotUsedInt",
        DSTBLK  := #SPtr
      );
NozHeaD:NOP   0;


REGION Network 28: **** 5.2 - Equations - Flow Equations **** Header DB's
   // Header
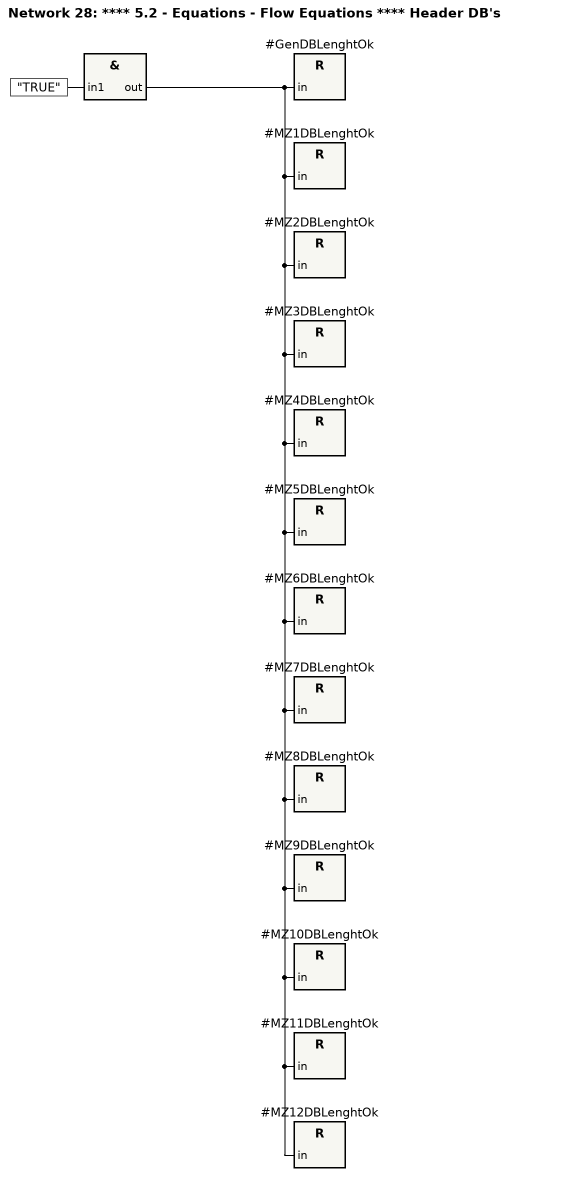
   IF "TRUE" THEN
       #GenDBLenghtOk := FALSE;
       #MZ1DBLenghtOk := FALSE;
       #MZ2DBLenghtOk := FALSE;
       #MZ3DBLenghtOk := FALSE;
       #MZ4DBLenghtOk := FALSE;
       #MZ5DBLenghtOk := FALSE;
       #MZ6DBLenghtOk := FALSE;
       #MZ7DBLenghtOk := FALSE;
       #MZ8DBLenghtOk := FALSE;
       #MZ9DBLenghtOk := FALSE;
       #MZ10DBLenghtOk := FALSE;
       #MZ11DBLenghtOk := FALSE;
       #MZ12DBLenghtOk := FALSE;
   END_IF;
END_REGION

NETWORK
TITLE = **** 5.2 - Equations - Flow Equations **** Header DB's
// Load Pointers For All Alarm DB:s


      OPN   #C_GenAlarmDB;  //General PLC Alarms
      L     DBLG;
      T     %DBW0;
      T     #GenDBLength;
      L     DBNO;
      T     #GenDBNumber;
      T     %DBW2;
      OPN   #C_GenAlarmCompare;  //General PLC Alarms
      L     DBLG;
      T     #GenDBLenghtCompare;
      L     #GenDBLength;
      L     #GenDBLenghtCompare;
      ==D;
      JCN   GenOk;
      L     #GenDBLenghtCompare;
      L     8;
      >=I;
      S     #GenDBLenghtOk;
GenOk:NOP   0;
      OPN   #C_AlarmDBMZ1;  // MZ Alarms
      L     DBLG;
      T     %DBW0;
      T     #MZ1DBLength;
      L     DBNO;
      T     #MZ1DBNumber;
      T     %DBW2;
      OPN   #C_AlarmCompareDBMZ1;  //MZ Alarms
      L     DBLG;
      T     #MZ1DBLenghtCompare;
      L     #MZ1DBLength;
      L     #MZ1DBLenghtCompare;
      ==D;
      JCN   MZ1Ok;
      L     #MZ1DBLenghtCompare;
      L     8;
      >=I;
      S     #MZ1DBLenghtOk;
MZ1Ok:NOP   0;
      OPN   #C_AlarmDBMZ2;  // MZ Alarms
      L     DBLG;
      T     %DBW0;
      T     #MZ2DBLength;
      L     DBNO;
      T     #MZ2DBNumber;
      T     %DBW2;
      OPN   #C_AlarmCompareDBMZ2;  //MZ Alarms
      L     DBLG;
      T     #MZ2DBLenghtCompare;
      L     #MZ2DBLength;
      L     #MZ2DBLenghtCompare;
      ==D;
      JCN   MZ2ok;
      L     #MZ2DBLenghtCompare;
      L     8;
      >=I;
      S     #MZ2DBLenghtOk;
MZ2ok:NOP   0;
      OPN   #C_AlarmDBMZ3;  // MZ Alarms
      L     DBLG;
      T     %DBW0;
      T     #MZ3DBLength;
      L     DBNO;
      T     #MZ3DBNumber;
      T     %DBW2;
      OPN   #C_AlarmCompareDBMZ3;  //MZ Alarms
      L     DBLG;
      T     #MZ3DBLenghtCompare;
      L     #MZ3DBLength;
      L     #MZ3DBLenghtCompare;
      ==D;
      JCN   MZ3ok;
      L     #MZ3DBLenghtCompare;
      L     8;
      >=I;
      S     #MZ3DBLenghtOk;
MZ3ok:NOP   0;
      OPN   #C_AlarmDBMZ4;  // MZ Alarms
      L     DBLG;
      T     %DBW0;
      T     #MZ4DBLength;
      L     DBNO;
      T     #MZ4DBNumber;
      T     %DBW2;
      OPN   #C_AlarmCompareDBMZ4;  //MZ Alarms
      L     DBLG;
      T     #MZ4DBLenghtCompare;
      L     #MZ4DBLength;
      L     #MZ4DBLenghtCompare;
      ==D;
      JCN   MZ4ok;
      L     #MZ4DBLenghtCompare;
      L     8;
      >=I;
      S     #MZ4DBLenghtOk;
MZ4ok:NOP   0;
      OPN   #C_AlarmDBMZ5;  // MZ Alarms
      L     DBLG;
      T     %DBW0;
      T     #MZ5DBLength;
      L     DBNO;
      T     #MZ5DBNumber;
      T     %DBW2;
      OPN   #C_AlarmCompareDBMZ5;  //MZ Alarms
      L     DBLG;
      T     #MZ5DBLenghtCompare;
      L     #MZ5DBLength;
      L     #MZ5DBLenghtCompare;
      ==D;
      JCN   MZ5ok;
      L     #MZ5DBLenghtCompare;
      L     8;
      >=I;
      S     #MZ5DBLenghtOk;
MZ5ok:NOP   0;
      OPN   #C_AlarmDBMZ6;  // MZ Alarms
      L     DBLG;
      T     %DBW0;
      T     #MZ6DBLength;
      L     DBNO;
      T     #MZ6DBNumber;
      T     %DBW2;
      OPN   #C_AlarmCompareDBMZ6;  //MZ Alarms
      L     DBLG;
      T     #MZ6DBLenghtCompare;
      L     #MZ6DBLength;
      L     #MZ6DBLenghtCompare;
      ==D;
      JCN   MZ6ok;
      L     #MZ6DBLenghtCompare;
      L     8;
      >=I;
      S     #MZ6DBLenghtOk;
MZ6ok:NOP   0;
      OPN   #C_AlarmDBMZ7;  // MZ Alarms
      L     DBLG;
      T     %DBW0;
      T     #MZ7DBLength;
      L     DBNO;
      T     #MZ7DBNumber;
      T     %DBW2;
      OPN   #C_AlarmCompareDBMZ7;  //MZ Alarms
      L     DBLG;
      T     #MZ7DBLenghtCompare;
      L     #MZ7DBLength;
      L     #MZ7DBLenghtCompare;
      ==D;
      JCN   MZ7ok;
      L     #MZ7DBLenghtCompare;
      L     8;
      >=I;
      S     #MZ7DBLenghtOk;
MZ7ok:NOP   0;
      OPN   #C_AlarmDBMZ8;  // MZ Alarms
      L     DBLG;
      T     %DBW0;
      T     #MZ8DBLength;
      L     DBNO;
      T     #MZ8DBNumber;
      T     %DBW2;
      OPN   #C_AlarmCompareDBMZ8;  //MZ Alarms
      L     DBLG;
      T     #MZ8DBLenghtCompare;
      L     #MZ8DBLength;
      L     #MZ8DBLenghtCompare;
      ==D;
      JCN   MZ8ok;
      L     #MZ8DBLenghtCompare;
      L     8;
      >=I;
      S     #MZ8DBLenghtOk;
MZ8ok:NOP   0;
      OPN   #C_AlarmDBMZ9;  // MZ Alarms
      L     DBLG;
      T     %DBW0;
      T     #MZ9DBLength;
      L     DBNO;
      T     #MZ9DBNumber;
      T     %DBW2;
      OPN   #C_AlarmCompareDBMZ9;  //MZ Alarms
      L     DBLG;
      T     #MZ9DBLenghtCompare;
      L     #MZ9DBLength;
      L     #MZ9DBLenghtCompare;
      ==D;
      JCN   MZ9ok;
      L     #MZ9DBLenghtCompare;
      L     8;
      >=I;
      S     #MZ9DBLenghtOk;
MZ9ok:NOP   0;
      OPN   #C_AlarmDBMZ10;  // MZ Alarms
      L     DBLG;
      T     %DBW0;
      T     #MZ10DBLength;
      L     DBNO;
      T     #MZ10DBNumber;
      T     %DBW2;
      OPN   #C_AlarmCompareDBMZ10;  //MZ Alarms
      L     DBLG;
      T     #MZ10DBLenghtCompare;
      L     #MZ10DBLength;
      L     #MZ10DBLenghtCompare;
      ==D;
      JCN   MZ10ok;
      L     #MZ10DBLenghtCompare;
      L     8;
      >=I;
      S     #MZ10DBLenghtOk;
MZ10ok:NOP   0;
      OPN   #C_AlarmDBMZ11;  // MZ Alarms
      L     DBLG;
      T     %DBW0;
      T     #MZ11DBLength;
      L     DBNO;
      T     #MZ11DBNumber;
      T     %DBW2;
      OPN   #C_AlarmCompareDBMZ11;  //MZ Alarms
      L     DBLG;
      T     #MZ11DBLenghtCompare;
      L     #MZ11DBLength;
      L     #MZ11DBLenghtCompare;
      ==D;
      JCN   MZ11ok;
      L     #MZ11DBLenghtCompare;
      L     8;
      >=I;
      S     #MZ11DBLenghtOk;
MZ11ok:NOP   0;
      OPN   #C_AlarmDBMZ12;  // MZ Alarms
      L     DBLG;
      T     %DBW0;
      T     #MZ12DBLength;
      L     DBNO;
      T     #MZ12DBNumber;
      OPN   #C_AlarmCompareDBMZ12;  //MZ Alarms
      L     DBLG;
      T     #MZ12DBLenghtCompare;
      L     #MZ12DBLength;
      L     #MZ12DBLenghtCompare;
      ==D;
      JCN   MZ12ok;
      L     #MZ12DBLenghtCompare;
      L     8;
      >=I;
      S     #MZ12DBLenghtOk;
MZ12ok:NOP   0;

      OPN   #C_AlarmDBMZ13;  // MZ Alarms
      L     DBLG;
      T     %DBW0;
      T     #MZ13DBLength;
      L     DBNO;
      T     #MZ13DBNumber;
      OPN   #C_AlarmCompareDBMZ13;  //MZ Alarms
      L     DBLG;
      T     #MZ13DBLenghtCompare;
      L     #MZ13DBLength;
      L     #MZ13DBLenghtCompare;
      ==D;
      JCN   MZ13ok;
      L     #MZ13DBLenghtCompare;
      L     8;
      >=I;
      S     #MZ13DBLenghtOk;

MZ13ok:NOP   0;

      OPN   #C_AlarmDBMZ14;  // MZ Alarms
      L     DBLG;
      T     %DBW0;
      T     #MZ14DBLength;
      L     DBNO;
      T     #MZ14DBNumber;
      OPN   #C_AlarmCompareDBMZ14;  //MZ Alarms
      L     DBLG;
      T     #MZ14DBLenghtCompare;
      L     #MZ14DBLength;
      L     #MZ14DBLenghtCompare;
      ==D;
      JCN   MZ14ok;
      L     #MZ14DBLenghtCompare;
      L     8;
      >=I;
      S     #MZ14DBLenghtOk;

MZ14ok:NOP   0;

//Alarm DB's Ok To Send
      A     #GenDBLenghtOk;
      =     #IO_AlarmDB.GenDBLenghtOk;
      A     #MZ1DBLenghtOk;
      =     #IO_AlarmDB.MZ1DBLenghtOk;
      A     #MZ2DBLenghtOk;
      =     #IO_AlarmDB.MZ2DBLenghtOk;
      A     #MZ3DBLenghtOk;
      =     #IO_AlarmDB.MZ3DBLenghtOk;
      A     #MZ4DBLenghtOk;
      =     #IO_AlarmDB.MZ4DBLenghtOk;
      A     #MZ5DBLenghtOk;
      =     #IO_AlarmDB.MZ5DBLenghtOk;
      A     #MZ6DBLenghtOk;
      =     #IO_AlarmDB.MZ6DBLenghtOk;
      A     #MZ7DBLenghtOk;
      =     #IO_AlarmDB.MZ7DBLenghtOk;
      A     #MZ8DBLenghtOk;
      =     #IO_AlarmDB.MZ8DBLenghtOk;
      A     #MZ9DBLenghtOk;
      =     #IO_AlarmDB.MZ9DBLenghtOk;
      A     #MZ10DBLenghtOk;
      =     #IO_AlarmDB.MZ10DBLenghtOk;
      A     #MZ11DBLenghtOk;
      =     #IO_AlarmDB.MZ11DBLenghtOk;
      A     #MZ12DBLenghtOk;
      =     #IO_AlarmDB.MZ12DBLenghtOk;
      A     #MZ13DBLenghtOk;
      =     #IO_AlarmDB.MZ13DBLenghtOk;
      A     #MZ14DBLenghtOk;
      =     #IO_AlarmDB.MZ14DBLenghtOk;

// Amount Of ModeZone
      L     #C_NbrOfModeZone;
      T     #IO_AlarmDB.C_NbrOfModeZone;


REGION Network 30: **** 5.2 - Flow Equations **** Filter
   // Filter
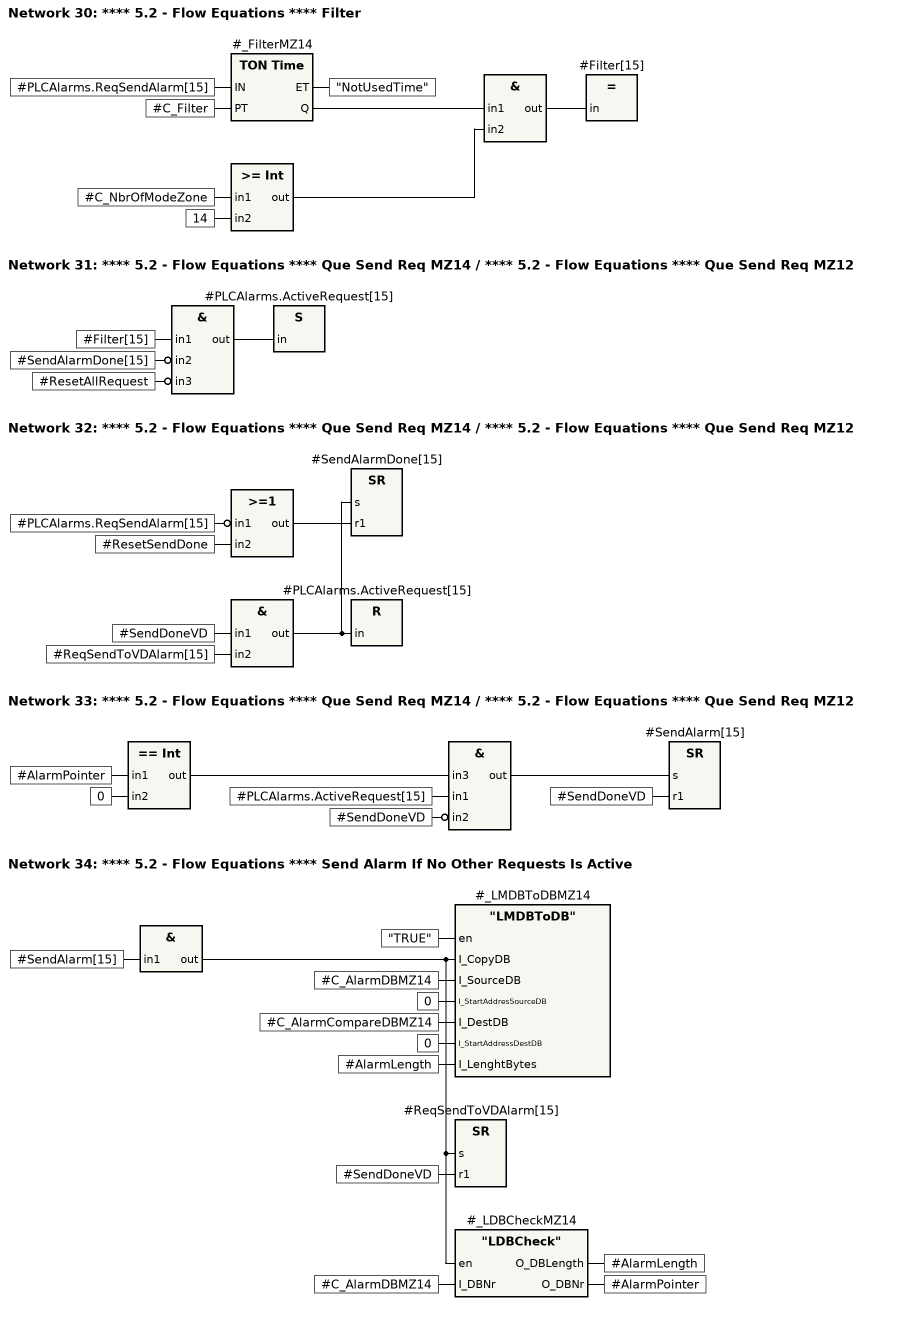
   #_FilterMZ14(IN := #PLCAlarms.ReqSendAlarm[15], PT := #C_Filter, ET => "NotUsedTime");   // TON
   #Filter[15] := #_FilterMZ14.Q AND (#C_NbrOfModeZone >= 14);
END_REGION

REGION Network 31: **** 5.2 - Flow Equations **** Que Send Req MZ14 / **** 5.2 - Flow Equations **** Que Send Req MZ12
   // Que Send Req
   IF #Filter[15] AND NOT #SendAlarmDone[15] AND NOT #ResetAllRequest THEN
       #PLCAlarms.ActiveRequest[15] := TRUE;
   END_IF;
END_REGION

REGION Network 32: **** 5.2 - Flow Equations **** Que Send Req MZ14 / **** 5.2 - Flow Equations **** Que Send Req MZ12
   // Que Send Req
   #_w1 := #SendDoneVD AND #ReqSendToVDAlarm[15];
   IF #_w1 THEN
       #SendAlarmDone[15] := TRUE;   // SR flip-flop
   END_IF;
   IF NOT #PLCAlarms.ReqSendAlarm[15] OR #ResetSendDone THEN #SendAlarmDone[15] := FALSE; END_IF;
   IF #_w1 THEN #PLCAlarms.ActiveRequest[15] := FALSE; END_IF;
END_REGION

REGION Network 33: **** 5.2 - Flow Equations **** Que Send Req MZ14 / **** 5.2 - Flow Equations **** Que Send Req MZ12
   // Que Send Req
   IF (#AlarmPointer = 0) AND #PLCAlarms.ActiveRequest[15] AND NOT #SendDoneVD THEN
       #SendAlarm[15] := TRUE;   // SR flip-flop
   END_IF;
   IF #SendDoneVD THEN #SendAlarm[15] := FALSE; END_IF;
END_REGION

REGION Network 34: **** 5.2 - Flow Equations **** Send Alarm If No Other Requests Is Active
   // Send Alarm If No Other Requests Is Active
   IF #SendAlarm[15] THEN
       #ReqSendToVDAlarm[15] := TRUE;   // SR flip-flop
   END_IF;
   IF #SendDoneVD THEN #ReqSendToVDAlarm[15] := FALSE; END_IF;
   IF #SendAlarm[15] THEN
       #_LDBCheckMZ14(I_DBNr := #C_AlarmDBMZ14, O_DBLength => #AlarmLength, O_DBNr => #AlarmPointer);   // "LDBCheck"
   END_IF;
   IF "TRUE" THEN
       #_LMDBToDBMZ14(I_CopyDB := #SendAlarm[15],   // "LMDBToDB"
                      I_SourceDB := #C_AlarmDBMZ14,
                      I_StartAddresSourceDB := 0,
                      I_DestDB := #C_AlarmCompareDBMZ14,
                      I_StartAddressDestDB := 0,
                      I_LenghtBytes := #AlarmLength);
   END_IF;
END_REGION

REGION Network 35: **** 5.2 - Flow Equations **** Filter
   // Filter
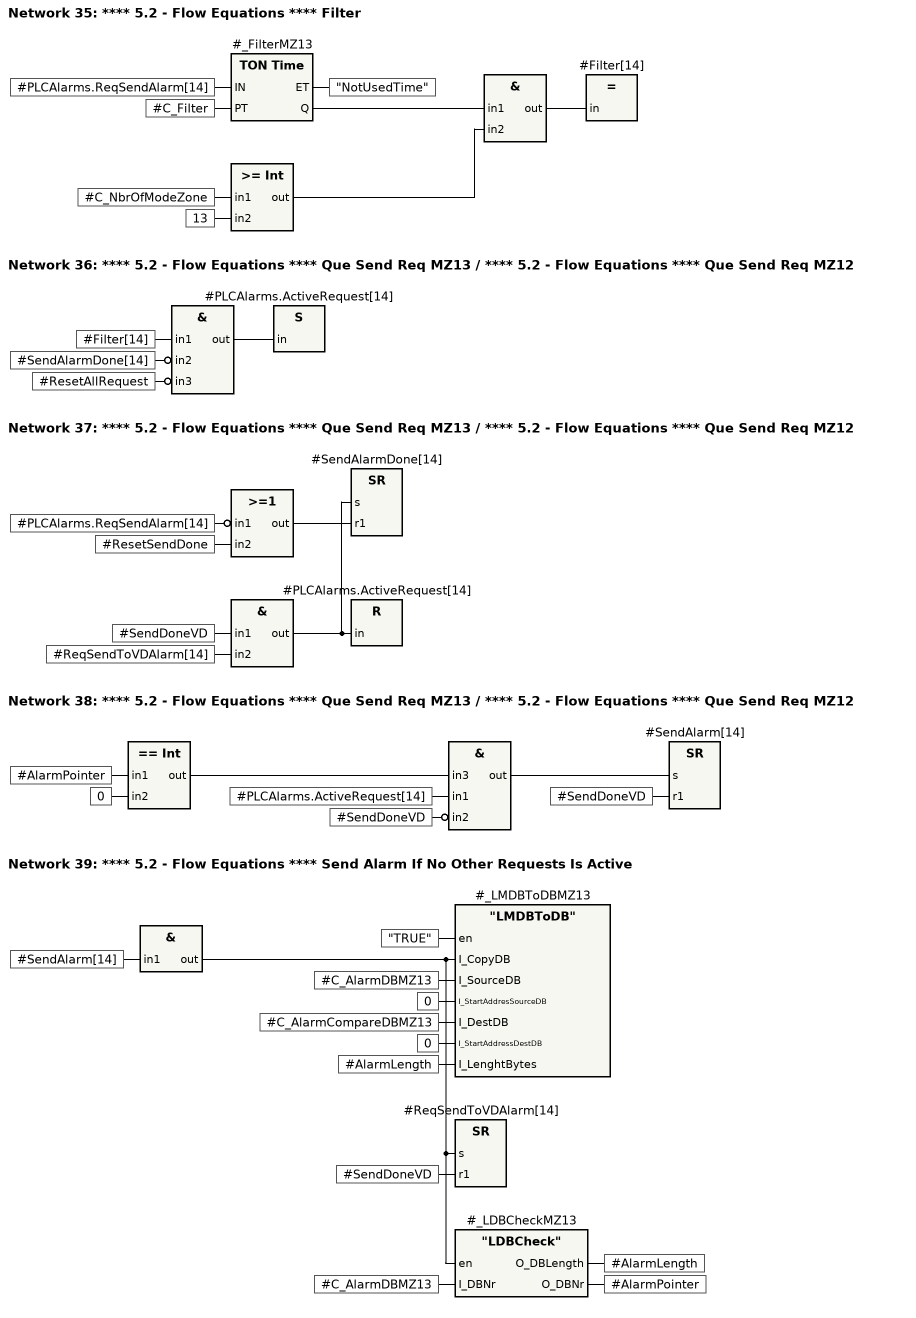
   #_FilterMZ13(IN := #PLCAlarms.ReqSendAlarm[14], PT := #C_Filter, ET => "NotUsedTime");   // TON
   #Filter[14] := #_FilterMZ13.Q AND (#C_NbrOfModeZone >= 13);
END_REGION

REGION Network 36: **** 5.2 - Flow Equations **** Que Send Req MZ13 / **** 5.2 - Flow Equations **** Que Send Req MZ12
   // Que Send Req
   IF #Filter[14] AND NOT #SendAlarmDone[14] AND NOT #ResetAllRequest THEN
       #PLCAlarms.ActiveRequest[14] := TRUE;
   END_IF;
END_REGION

REGION Network 37: **** 5.2 - Flow Equations **** Que Send Req MZ13 / **** 5.2 - Flow Equations **** Que Send Req MZ12
   // Que Send Req
   #_w1 := #SendDoneVD AND #ReqSendToVDAlarm[14];
   IF #_w1 THEN
       #SendAlarmDone[14] := TRUE;   // SR flip-flop
   END_IF;
   IF NOT #PLCAlarms.ReqSendAlarm[14] OR #ResetSendDone THEN #SendAlarmDone[14] := FALSE; END_IF;
   IF #_w1 THEN #PLCAlarms.ActiveRequest[14] := FALSE; END_IF;
END_REGION

REGION Network 38: **** 5.2 - Flow Equations **** Que Send Req MZ13 / **** 5.2 - Flow Equations **** Que Send Req MZ12
   // Que Send Req
   IF (#AlarmPointer = 0) AND #PLCAlarms.ActiveRequest[14] AND NOT #SendDoneVD THEN
       #SendAlarm[14] := TRUE;   // SR flip-flop
   END_IF;
   IF #SendDoneVD THEN #SendAlarm[14] := FALSE; END_IF;
END_REGION

REGION Network 39: **** 5.2 - Flow Equations **** Send Alarm If No Other Requests Is Active
   // Send Alarm If No Other Requests Is Active
   IF #SendAlarm[14] THEN
       #ReqSendToVDAlarm[14] := TRUE;   // SR flip-flop
   END_IF;
   IF #SendDoneVD THEN #ReqSendToVDAlarm[14] := FALSE; END_IF;
   IF #SendAlarm[14] THEN
       #_LDBCheckMZ13(I_DBNr := #C_AlarmDBMZ13, O_DBLength => #AlarmLength, O_DBNr => #AlarmPointer);   // "LDBCheck"
   END_IF;
   IF "TRUE" THEN
       #_LMDBToDBMZ13(I_CopyDB := #SendAlarm[14],   // "LMDBToDB"
                      I_SourceDB := #C_AlarmDBMZ13,
                      I_StartAddresSourceDB := 0,
                      I_DestDB := #C_AlarmCompareDBMZ13,
                      I_StartAddressDestDB := 0,
                      I_LenghtBytes := #AlarmLength);
   END_IF;
END_REGION

REGION Network 40: **** 5.2 - Flow Equations **** Filter
   // Filter
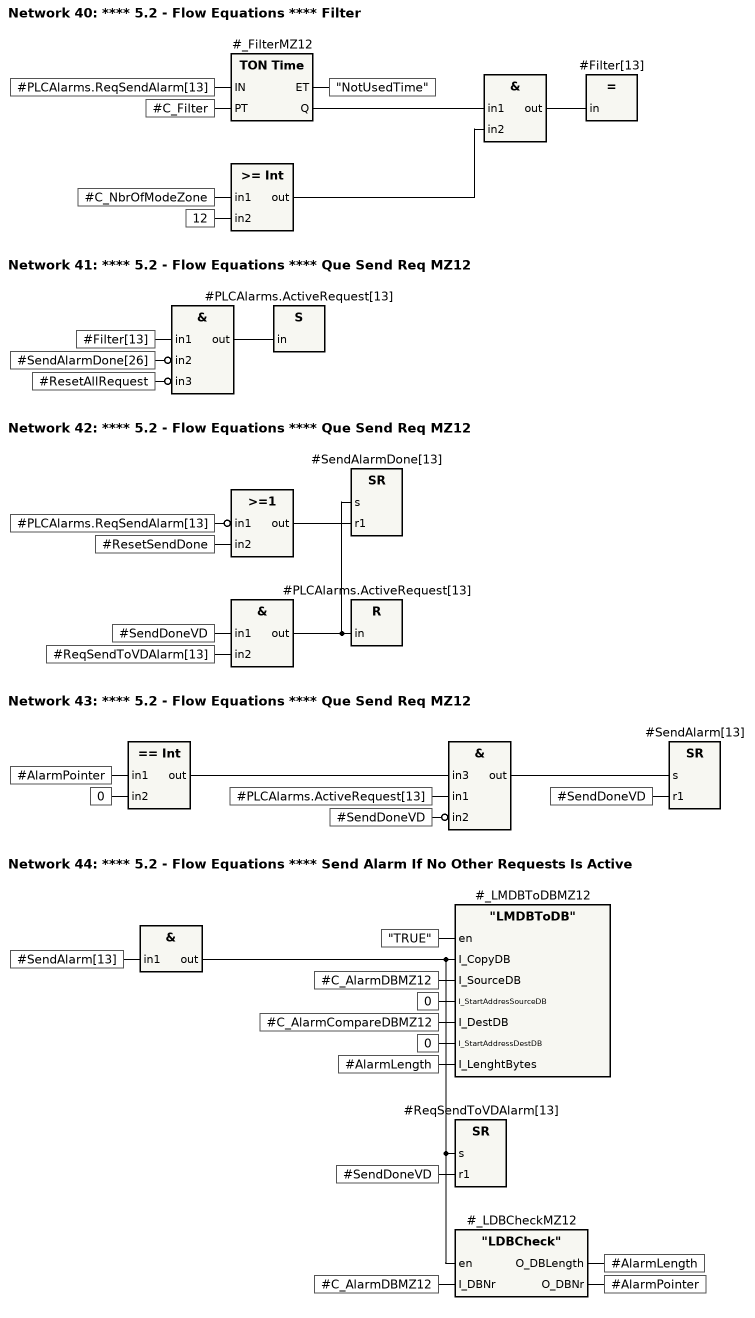
   #_FilterMZ12(IN := #PLCAlarms.ReqSendAlarm[13], PT := #C_Filter, ET => "NotUsedTime");   // TON
   #Filter[13] := #_FilterMZ12.Q AND (#C_NbrOfModeZone >= 12);
END_REGION

REGION Network 41: **** 5.2 - Flow Equations **** Que Send Req MZ12
   // Que Send Req
   IF #Filter[13] AND NOT #SendAlarmDone[26] AND NOT #ResetAllRequest THEN
       #PLCAlarms.ActiveRequest[13] := TRUE;
   END_IF;
END_REGION

REGION Network 42: **** 5.2 - Flow Equations **** Que Send Req MZ12
   // Que Send Req
   #_w1 := #SendDoneVD AND #ReqSendToVDAlarm[13];
   IF #_w1 THEN
       #SendAlarmDone[13] := TRUE;   // SR flip-flop
   END_IF;
   IF NOT #PLCAlarms.ReqSendAlarm[13] OR #ResetSendDone THEN #SendAlarmDone[13] := FALSE; END_IF;
   IF #_w1 THEN #PLCAlarms.ActiveRequest[13] := FALSE; END_IF;
END_REGION

REGION Network 43: **** 5.2 - Flow Equations **** Que Send Req MZ12
   // Que Send Req
   IF (#AlarmPointer = 0) AND #PLCAlarms.ActiveRequest[13] AND NOT #SendDoneVD THEN
       #SendAlarm[13] := TRUE;   // SR flip-flop
   END_IF;
   IF #SendDoneVD THEN #SendAlarm[13] := FALSE; END_IF;
END_REGION

REGION Network 44: **** 5.2 - Flow Equations **** Send Alarm If No Other Requests Is Active
   // Send Alarm If No Other Requests Is Active
   IF #SendAlarm[13] THEN
       #ReqSendToVDAlarm[13] := TRUE;   // SR flip-flop
   END_IF;
   IF #SendDoneVD THEN #ReqSendToVDAlarm[13] := FALSE; END_IF;
   IF #SendAlarm[13] THEN
       #_LDBCheckMZ12(I_DBNr := #C_AlarmDBMZ12, O_DBLength => #AlarmLength, O_DBNr => #AlarmPointer);   // "LDBCheck"
   END_IF;
   IF "TRUE" THEN
       #_LMDBToDBMZ12(I_CopyDB := #SendAlarm[13],   // "LMDBToDB"
                      I_SourceDB := #C_AlarmDBMZ12,
                      I_StartAddresSourceDB := 0,
                      I_DestDB := #C_AlarmCompareDBMZ12,
                      I_StartAddressDestDB := 0,
                      I_LenghtBytes := #AlarmLength);
   END_IF;
END_REGION

REGION Network 45: **** 5.2 - Flow Equations **** Filter
   // Filter
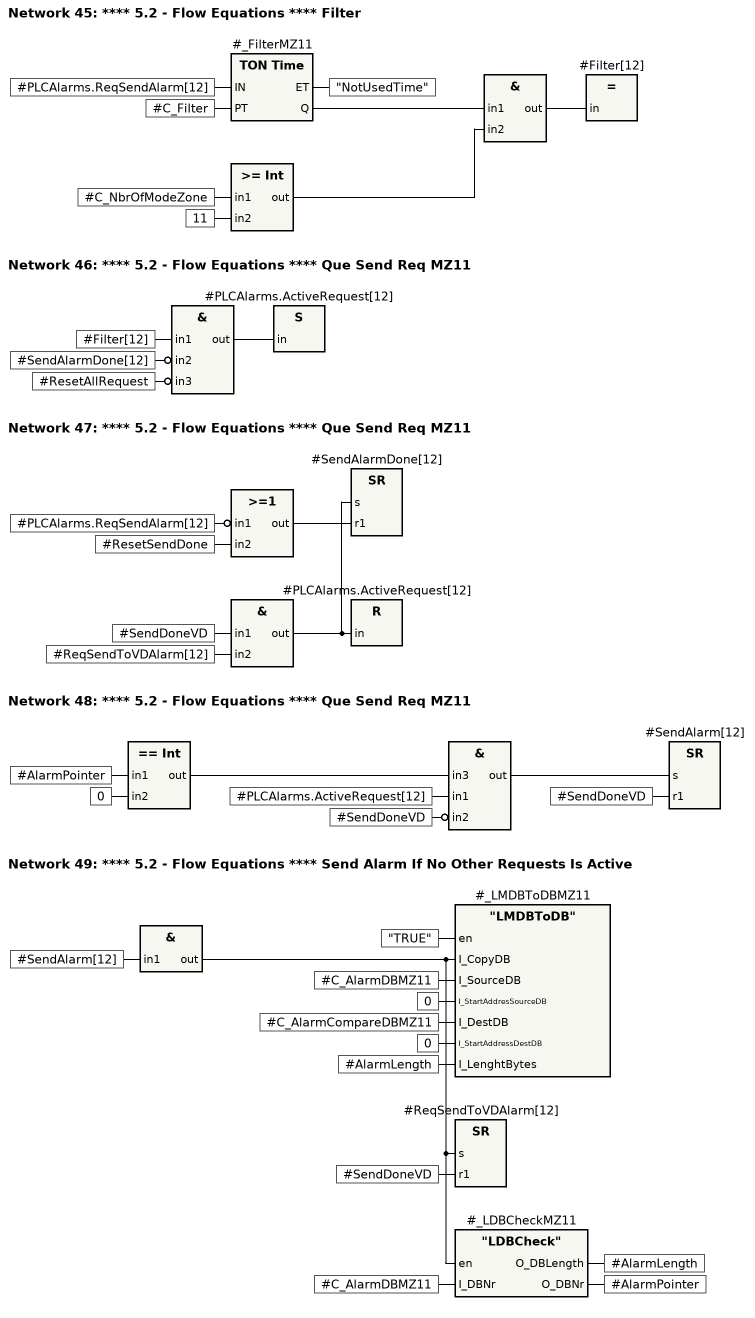
   #_FilterMZ11(IN := #PLCAlarms.ReqSendAlarm[12], PT := #C_Filter, ET => "NotUsedTime");   // TON
   #Filter[12] := #_FilterMZ11.Q AND (#C_NbrOfModeZone >= 11);
END_REGION

REGION Network 46: **** 5.2 - Flow Equations **** Que Send Req MZ11
   // Que Send Req
   IF #Filter[12] AND NOT #SendAlarmDone[12] AND NOT #ResetAllRequest THEN
       #PLCAlarms.ActiveRequest[12] := TRUE;
   END_IF;
END_REGION

REGION Network 47: **** 5.2 - Flow Equations **** Que Send Req MZ11
   // Que Send Req
   #_w1 := #SendDoneVD AND #ReqSendToVDAlarm[12];
   IF #_w1 THEN
       #SendAlarmDone[12] := TRUE;   // SR flip-flop
   END_IF;
   IF NOT #PLCAlarms.ReqSendAlarm[12] OR #ResetSendDone THEN #SendAlarmDone[12] := FALSE; END_IF;
   IF #_w1 THEN #PLCAlarms.ActiveRequest[12] := FALSE; END_IF;
END_REGION

REGION Network 48: **** 5.2 - Flow Equations **** Que Send Req MZ11
   // Que Send Req
   IF (#AlarmPointer = 0) AND #PLCAlarms.ActiveRequest[12] AND NOT #SendDoneVD THEN
       #SendAlarm[12] := TRUE;   // SR flip-flop
   END_IF;
   IF #SendDoneVD THEN #SendAlarm[12] := FALSE; END_IF;
END_REGION

REGION Network 49: **** 5.2 - Flow Equations **** Send Alarm If No Other Requests Is Active
   // Send Alarm If No Other Requests Is Active
   IF #SendAlarm[12] THEN
       #ReqSendToVDAlarm[12] := TRUE;   // SR flip-flop
   END_IF;
   IF #SendDoneVD THEN #ReqSendToVDAlarm[12] := FALSE; END_IF;
   IF #SendAlarm[12] THEN
       #_LDBCheckMZ11(I_DBNr := #C_AlarmDBMZ11, O_DBLength => #AlarmLength, O_DBNr => #AlarmPointer);   // "LDBCheck"
   END_IF;
   IF "TRUE" THEN
       #_LMDBToDBMZ11(I_CopyDB := #SendAlarm[12],   // "LMDBToDB"
                      I_SourceDB := #C_AlarmDBMZ11,
                      I_StartAddresSourceDB := 0,
                      I_DestDB := #C_AlarmCompareDBMZ11,
                      I_StartAddressDestDB := 0,
                      I_LenghtBytes := #AlarmLength);
   END_IF;
END_REGION

REGION Network 50: **** 5.2 - Flow Equations **** Filter
   // Filter
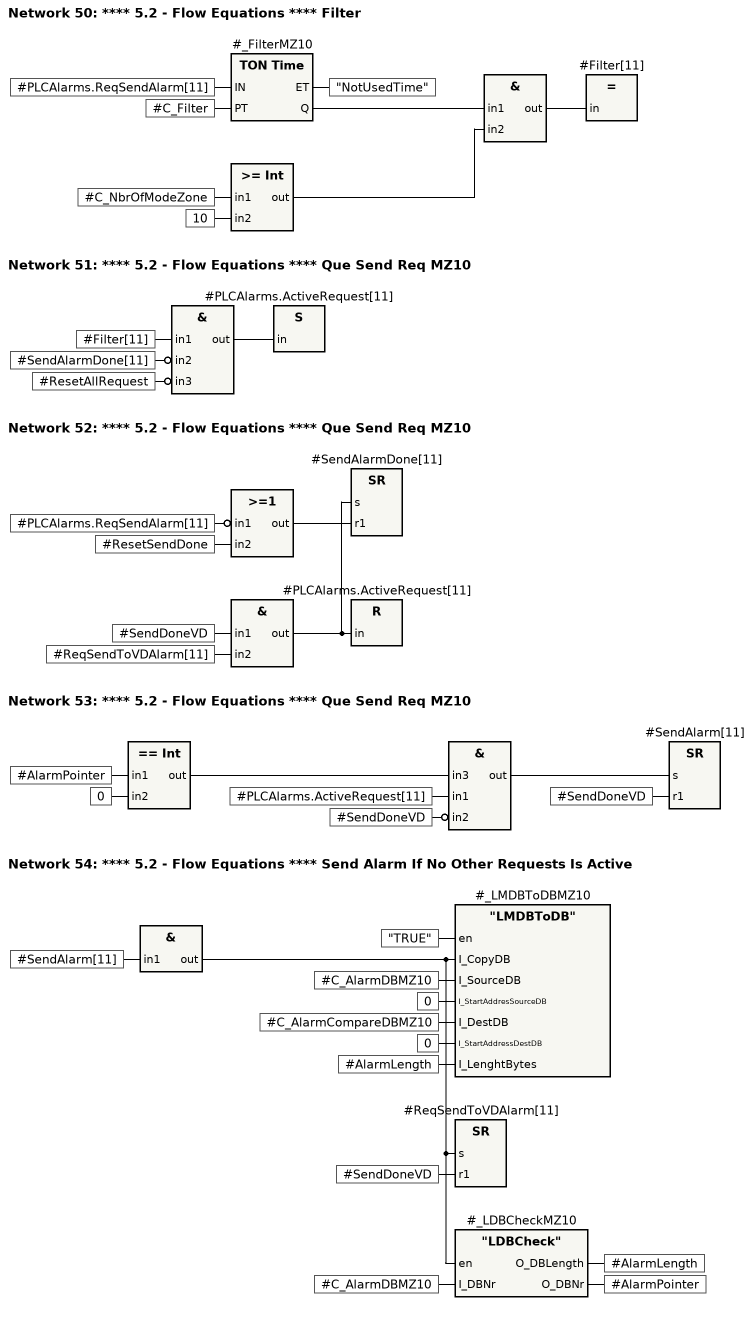
   #_FilterMZ10(IN := #PLCAlarms.ReqSendAlarm[11], PT := #C_Filter, ET => "NotUsedTime");   // TON
   #Filter[11] := #_FilterMZ10.Q AND (#C_NbrOfModeZone >= 10);
END_REGION

REGION Network 51: **** 5.2 - Flow Equations **** Que Send Req MZ10
   // Que Send Req
   IF #Filter[11] AND NOT #SendAlarmDone[11] AND NOT #ResetAllRequest THEN
       #PLCAlarms.ActiveRequest[11] := TRUE;
   END_IF;
END_REGION

REGION Network 52: **** 5.2 - Flow Equations **** Que Send Req MZ10
   // Que Send Req
   #_w1 := #SendDoneVD AND #ReqSendToVDAlarm[11];
   IF #_w1 THEN
       #SendAlarmDone[11] := TRUE;   // SR flip-flop
   END_IF;
   IF NOT #PLCAlarms.ReqSendAlarm[11] OR #ResetSendDone THEN #SendAlarmDone[11] := FALSE; END_IF;
   IF #_w1 THEN #PLCAlarms.ActiveRequest[11] := FALSE; END_IF;
END_REGION

REGION Network 53: **** 5.2 - Flow Equations **** Que Send Req MZ10
   // Que Send Req
   IF (#AlarmPointer = 0) AND #PLCAlarms.ActiveRequest[11] AND NOT #SendDoneVD THEN
       #SendAlarm[11] := TRUE;   // SR flip-flop
   END_IF;
   IF #SendDoneVD THEN #SendAlarm[11] := FALSE; END_IF;
END_REGION

REGION Network 54: **** 5.2 - Flow Equations **** Send Alarm If No Other Requests Is Active
   // Send Alarm If No Other Requests Is Active
   IF #SendAlarm[11] THEN
       #ReqSendToVDAlarm[11] := TRUE;   // SR flip-flop
   END_IF;
   IF #SendDoneVD THEN #ReqSendToVDAlarm[11] := FALSE; END_IF;
   IF #SendAlarm[11] THEN
       #_LDBCheckMZ10(I_DBNr := #C_AlarmDBMZ10, O_DBLength => #AlarmLength, O_DBNr => #AlarmPointer);   // "LDBCheck"
   END_IF;
   IF "TRUE" THEN
       #_LMDBToDBMZ10(I_CopyDB := #SendAlarm[11],   // "LMDBToDB"
                      I_SourceDB := #C_AlarmDBMZ10,
                      I_StartAddresSourceDB := 0,
                      I_DestDB := #C_AlarmCompareDBMZ10,
                      I_StartAddressDestDB := 0,
                      I_LenghtBytes := #AlarmLength);
   END_IF;
END_REGION

REGION Network 55: **** 5.2 - Flow Equations **** Filter
   // Filter
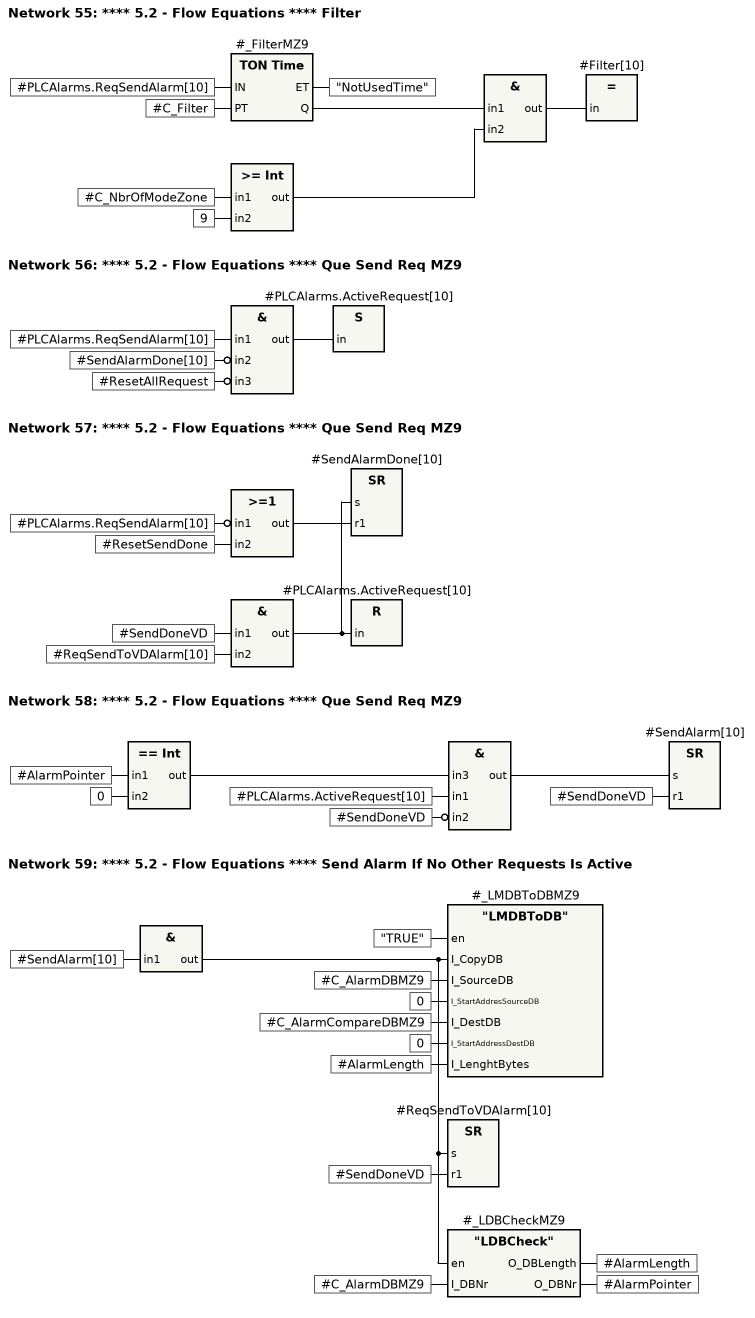
   #_FilterMZ9(IN := #PLCAlarms.ReqSendAlarm[10], PT := #C_Filter, ET => "NotUsedTime");   // TON
   #Filter[10] := #_FilterMZ9.Q AND (#C_NbrOfModeZone >= 9);
END_REGION

REGION Network 56: **** 5.2 - Flow Equations **** Que Send Req MZ9
   // Que Send Req
   IF #PLCAlarms.ReqSendAlarm[10] AND NOT #SendAlarmDone[10] AND NOT #ResetAllRequest THEN
       #PLCAlarms.ActiveRequest[10] := TRUE;
   END_IF;
END_REGION

REGION Network 57: **** 5.2 - Flow Equations **** Que Send Req MZ9
   // Que Send Req
   #_w1 := #SendDoneVD AND #ReqSendToVDAlarm[10];
   IF #_w1 THEN
       #SendAlarmDone[10] := TRUE;   // SR flip-flop
   END_IF;
   IF NOT #PLCAlarms.ReqSendAlarm[10] OR #ResetSendDone THEN #SendAlarmDone[10] := FALSE; END_IF;
   IF #_w1 THEN #PLCAlarms.ActiveRequest[10] := FALSE; END_IF;
END_REGION

REGION Network 58: **** 5.2 - Flow Equations **** Que Send Req MZ9
   // Que Send Req
   IF (#AlarmPointer = 0) AND #PLCAlarms.ActiveRequest[10] AND NOT #SendDoneVD THEN
       #SendAlarm[10] := TRUE;   // SR flip-flop
   END_IF;
   IF #SendDoneVD THEN #SendAlarm[10] := FALSE; END_IF;
END_REGION

REGION Network 59: **** 5.2 - Flow Equations **** Send Alarm If No Other Requests Is Active
   // Send Alarm If No Other Requests Is Active
   IF #SendAlarm[10] THEN
       #ReqSendToVDAlarm[10] := TRUE;   // SR flip-flop
   END_IF;
   IF #SendDoneVD THEN #ReqSendToVDAlarm[10] := FALSE; END_IF;
   IF #SendAlarm[10] THEN
       #_LDBCheckMZ9(I_DBNr := #C_AlarmDBMZ9, O_DBLength => #AlarmLength, O_DBNr => #AlarmPointer);   // "LDBCheck"
   END_IF;
   IF "TRUE" THEN
       #_LMDBToDBMZ9(I_CopyDB := #SendAlarm[10],   // "LMDBToDB"
                     I_SourceDB := #C_AlarmDBMZ9,
                     I_StartAddresSourceDB := 0,
                     I_DestDB := #C_AlarmCompareDBMZ9,
                     I_StartAddressDestDB := 0,
                     I_LenghtBytes := #AlarmLength);
   END_IF;
END_REGION

REGION Network 60: **** 5.2 - Flow Equations **** Filter
   // Filter
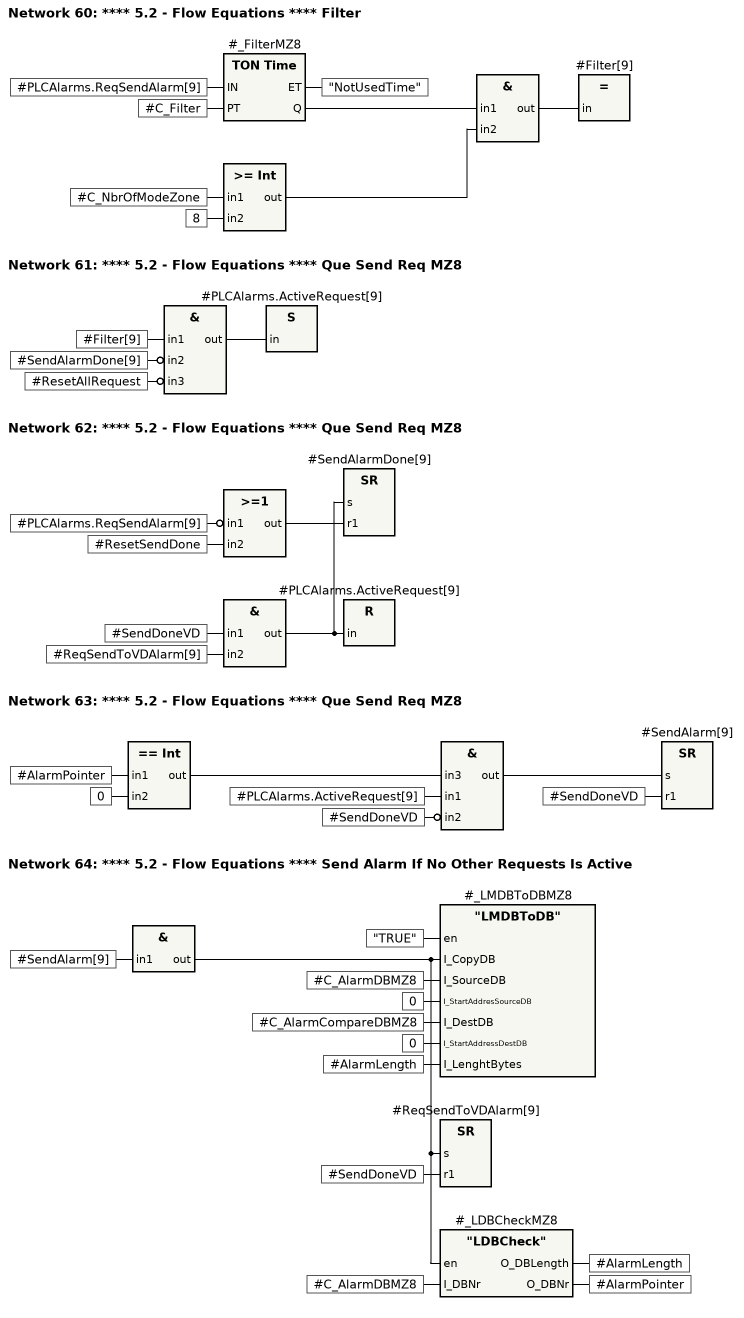
   #_FilterMZ8(IN := #PLCAlarms.ReqSendAlarm[9], PT := #C_Filter, ET => "NotUsedTime");   // TON
   #Filter[9] := #_FilterMZ8.Q AND (#C_NbrOfModeZone >= 8);
END_REGION

REGION Network 61: **** 5.2 - Flow Equations **** Que Send Req MZ8
   // Que Send Req
   IF #Filter[9] AND NOT #SendAlarmDone[9] AND NOT #ResetAllRequest THEN
       #PLCAlarms.ActiveRequest[9] := TRUE;
   END_IF;
END_REGION

REGION Network 62: **** 5.2 - Flow Equations **** Que Send Req MZ8
   // Que Send Req
   #_w1 := #SendDoneVD AND #ReqSendToVDAlarm[9];
   IF #_w1 THEN
       #SendAlarmDone[9] := TRUE;   // SR flip-flop
   END_IF;
   IF NOT #PLCAlarms.ReqSendAlarm[9] OR #ResetSendDone THEN #SendAlarmDone[9] := FALSE; END_IF;
   IF #_w1 THEN #PLCAlarms.ActiveRequest[9] := FALSE; END_IF;
END_REGION

REGION Network 63: **** 5.2 - Flow Equations **** Que Send Req MZ8
   // Que Send Req
   IF (#AlarmPointer = 0) AND #PLCAlarms.ActiveRequest[9] AND NOT #SendDoneVD THEN
       #SendAlarm[9] := TRUE;   // SR flip-flop
   END_IF;
   IF #SendDoneVD THEN #SendAlarm[9] := FALSE; END_IF;
END_REGION

REGION Network 64: **** 5.2 - Flow Equations **** Send Alarm If No Other Requests Is Active
   // Send Alarm If No Other Requests Is Active
   IF #SendAlarm[9] THEN
       #ReqSendToVDAlarm[9] := TRUE;   // SR flip-flop
   END_IF;
   IF #SendDoneVD THEN #ReqSendToVDAlarm[9] := FALSE; END_IF;
   IF #SendAlarm[9] THEN
       #_LDBCheckMZ8(I_DBNr := #C_AlarmDBMZ8, O_DBLength => #AlarmLength, O_DBNr => #AlarmPointer);   // "LDBCheck"
   END_IF;
   IF "TRUE" THEN
       #_LMDBToDBMZ8(I_CopyDB := #SendAlarm[9],   // "LMDBToDB"
                     I_SourceDB := #C_AlarmDBMZ8,
                     I_StartAddresSourceDB := 0,
                     I_DestDB := #C_AlarmCompareDBMZ8,
                     I_StartAddressDestDB := 0,
                     I_LenghtBytes := #AlarmLength);
   END_IF;
END_REGION

REGION Network 65: **** 5.2 - Flow Equations **** Filter
   // Filter
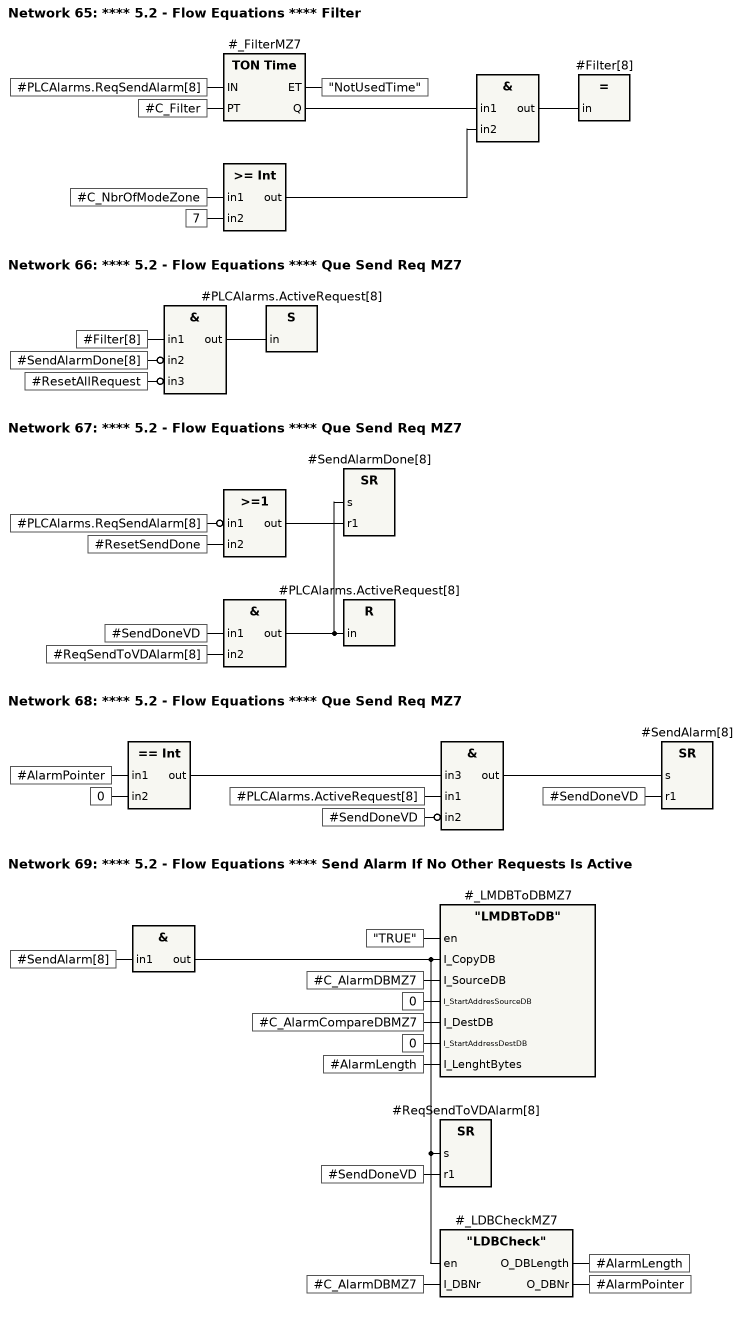
   #_FilterMZ7(IN := #PLCAlarms.ReqSendAlarm[8], PT := #C_Filter, ET => "NotUsedTime");   // TON
   #Filter[8] := #_FilterMZ7.Q AND (#C_NbrOfModeZone >= 7);
END_REGION

REGION Network 66: **** 5.2 - Flow Equations **** Que Send Req MZ7
   // Que Send Req
   IF #Filter[8] AND NOT #SendAlarmDone[8] AND NOT #ResetAllRequest THEN
       #PLCAlarms.ActiveRequest[8] := TRUE;
   END_IF;
END_REGION

REGION Network 67: **** 5.2 - Flow Equations **** Que Send Req MZ7
   // Que Send Req
   #_w1 := #SendDoneVD AND #ReqSendToVDAlarm[8];
   IF #_w1 THEN
       #SendAlarmDone[8] := TRUE;   // SR flip-flop
   END_IF;
   IF NOT #PLCAlarms.ReqSendAlarm[8] OR #ResetSendDone THEN #SendAlarmDone[8] := FALSE; END_IF;
   IF #_w1 THEN #PLCAlarms.ActiveRequest[8] := FALSE; END_IF;
END_REGION

REGION Network 68: **** 5.2 - Flow Equations **** Que Send Req MZ7
   // Que Send Req
   IF (#AlarmPointer = 0) AND #PLCAlarms.ActiveRequest[8] AND NOT #SendDoneVD THEN
       #SendAlarm[8] := TRUE;   // SR flip-flop
   END_IF;
   IF #SendDoneVD THEN #SendAlarm[8] := FALSE; END_IF;
END_REGION

REGION Network 69: **** 5.2 - Flow Equations **** Send Alarm If No Other Requests Is Active
   // Send Alarm If No Other Requests Is Active
   IF #SendAlarm[8] THEN
       #ReqSendToVDAlarm[8] := TRUE;   // SR flip-flop
   END_IF;
   IF #SendDoneVD THEN #ReqSendToVDAlarm[8] := FALSE; END_IF;
   IF #SendAlarm[8] THEN
       #_LDBCheckMZ7(I_DBNr := #C_AlarmDBMZ7, O_DBLength => #AlarmLength, O_DBNr => #AlarmPointer);   // "LDBCheck"
   END_IF;
   IF "TRUE" THEN
       #_LMDBToDBMZ7(I_CopyDB := #SendAlarm[8],   // "LMDBToDB"
                     I_SourceDB := #C_AlarmDBMZ7,
                     I_StartAddresSourceDB := 0,
                     I_DestDB := #C_AlarmCompareDBMZ7,
                     I_StartAddressDestDB := 0,
                     I_LenghtBytes := #AlarmLength);
   END_IF;
END_REGION

REGION Network 70: **** 5.2 - Flow Equations **** Filter
   // Filter
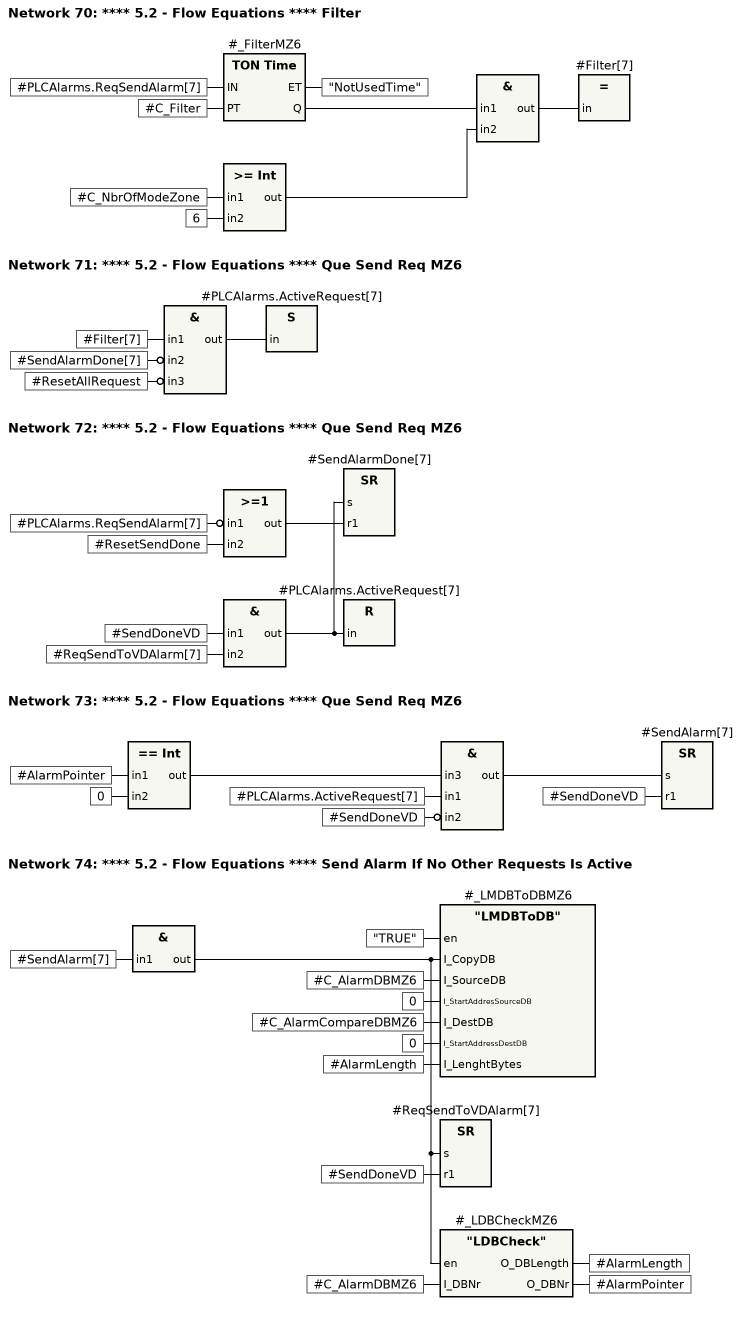
   #_FilterMZ6(IN := #PLCAlarms.ReqSendAlarm[7], PT := #C_Filter, ET => "NotUsedTime");   // TON
   #Filter[7] := #_FilterMZ6.Q AND (#C_NbrOfModeZone >= 6);
END_REGION

REGION Network 71: **** 5.2 - Flow Equations **** Que Send Req MZ6
   // Que Send Req
   IF #Filter[7] AND NOT #SendAlarmDone[7] AND NOT #ResetAllRequest THEN
       #PLCAlarms.ActiveRequest[7] := TRUE;
   END_IF;
END_REGION

REGION Network 72: **** 5.2 - Flow Equations **** Que Send Req MZ6
   // Que Send Req
   #_w1 := #SendDoneVD AND #ReqSendToVDAlarm[7];
   IF #_w1 THEN
       #SendAlarmDone[7] := TRUE;   // SR flip-flop
   END_IF;
   IF NOT #PLCAlarms.ReqSendAlarm[7] OR #ResetSendDone THEN #SendAlarmDone[7] := FALSE; END_IF;
   IF #_w1 THEN #PLCAlarms.ActiveRequest[7] := FALSE; END_IF;
END_REGION

REGION Network 73: **** 5.2 - Flow Equations **** Que Send Req MZ6
   // Que Send Req
   IF (#AlarmPointer = 0) AND #PLCAlarms.ActiveRequest[7] AND NOT #SendDoneVD THEN
       #SendAlarm[7] := TRUE;   // SR flip-flop
   END_IF;
   IF #SendDoneVD THEN #SendAlarm[7] := FALSE; END_IF;
END_REGION

REGION Network 74: **** 5.2 - Flow Equations **** Send Alarm If No Other Requests Is Active
   // Send Alarm If No Other Requests Is Active
   IF #SendAlarm[7] THEN
       #ReqSendToVDAlarm[7] := TRUE;   // SR flip-flop
   END_IF;
   IF #SendDoneVD THEN #ReqSendToVDAlarm[7] := FALSE; END_IF;
   IF #SendAlarm[7] THEN
       #_LDBCheckMZ6(I_DBNr := #C_AlarmDBMZ6, O_DBLength => #AlarmLength, O_DBNr => #AlarmPointer);   // "LDBCheck"
   END_IF;
   IF "TRUE" THEN
       #_LMDBToDBMZ6(I_CopyDB := #SendAlarm[7],   // "LMDBToDB"
                     I_SourceDB := #C_AlarmDBMZ6,
                     I_StartAddresSourceDB := 0,
                     I_DestDB := #C_AlarmCompareDBMZ6,
                     I_StartAddressDestDB := 0,
                     I_LenghtBytes := #AlarmLength);
   END_IF;
END_REGION

REGION Network 75: **** 5.2 - Flow Equations **** Filter
   // Filter
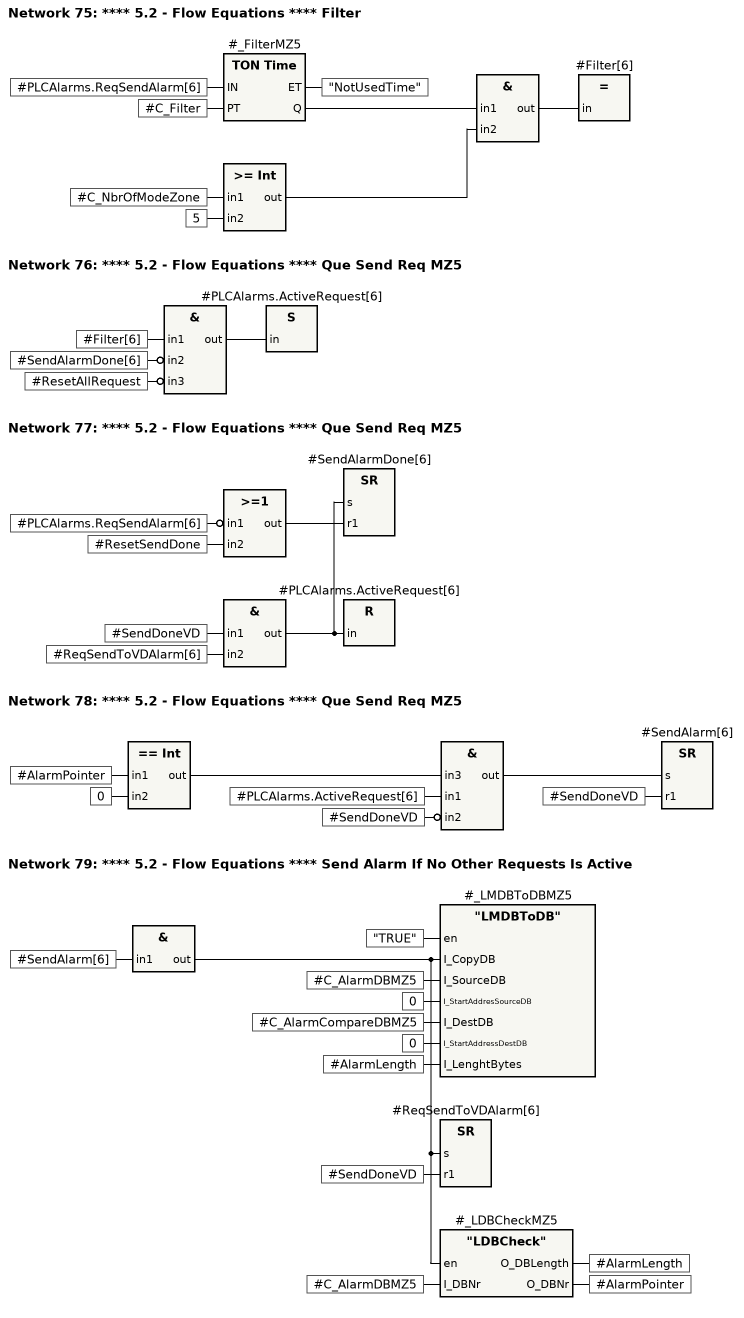
   #_FilterMZ5(IN := #PLCAlarms.ReqSendAlarm[6], PT := #C_Filter, ET => "NotUsedTime");   // TON
   #Filter[6] := #_FilterMZ5.Q AND (#C_NbrOfModeZone >= 5);
END_REGION

REGION Network 76: **** 5.2 - Flow Equations **** Que Send Req MZ5
   // Que Send Req
   IF #Filter[6] AND NOT #SendAlarmDone[6] AND NOT #ResetAllRequest THEN
       #PLCAlarms.ActiveRequest[6] := TRUE;
   END_IF;
END_REGION

REGION Network 77: **** 5.2 - Flow Equations **** Que Send Req MZ5
   // Que Send Req
   #_w1 := #SendDoneVD AND #ReqSendToVDAlarm[6];
   IF #_w1 THEN
       #SendAlarmDone[6] := TRUE;   // SR flip-flop
   END_IF;
   IF NOT #PLCAlarms.ReqSendAlarm[6] OR #ResetSendDone THEN #SendAlarmDone[6] := FALSE; END_IF;
   IF #_w1 THEN #PLCAlarms.ActiveRequest[6] := FALSE; END_IF;
END_REGION

REGION Network 78: **** 5.2 - Flow Equations **** Que Send Req MZ5
   // Que Send Req
   IF (#AlarmPointer = 0) AND #PLCAlarms.ActiveRequest[6] AND NOT #SendDoneVD THEN
       #SendAlarm[6] := TRUE;   // SR flip-flop
   END_IF;
   IF #SendDoneVD THEN #SendAlarm[6] := FALSE; END_IF;
END_REGION

REGION Network 79: **** 5.2 - Flow Equations **** Send Alarm If No Other Requests Is Active
   // Send Alarm If No Other Requests Is Active
   IF #SendAlarm[6] THEN
       #ReqSendToVDAlarm[6] := TRUE;   // SR flip-flop
   END_IF;
   IF #SendDoneVD THEN #ReqSendToVDAlarm[6] := FALSE; END_IF;
   IF #SendAlarm[6] THEN
       #_LDBCheckMZ5(I_DBNr := #C_AlarmDBMZ5, O_DBLength => #AlarmLength, O_DBNr => #AlarmPointer);   // "LDBCheck"
   END_IF;
   IF "TRUE" THEN
       #_LMDBToDBMZ5(I_CopyDB := #SendAlarm[6],   // "LMDBToDB"
                     I_SourceDB := #C_AlarmDBMZ5,
                     I_StartAddresSourceDB := 0,
                     I_DestDB := #C_AlarmCompareDBMZ5,
                     I_StartAddressDestDB := 0,
                     I_LenghtBytes := #AlarmLength);
   END_IF;
END_REGION

REGION Network 80: **** 5.2 - Flow Equations **** Filter
   // Filter
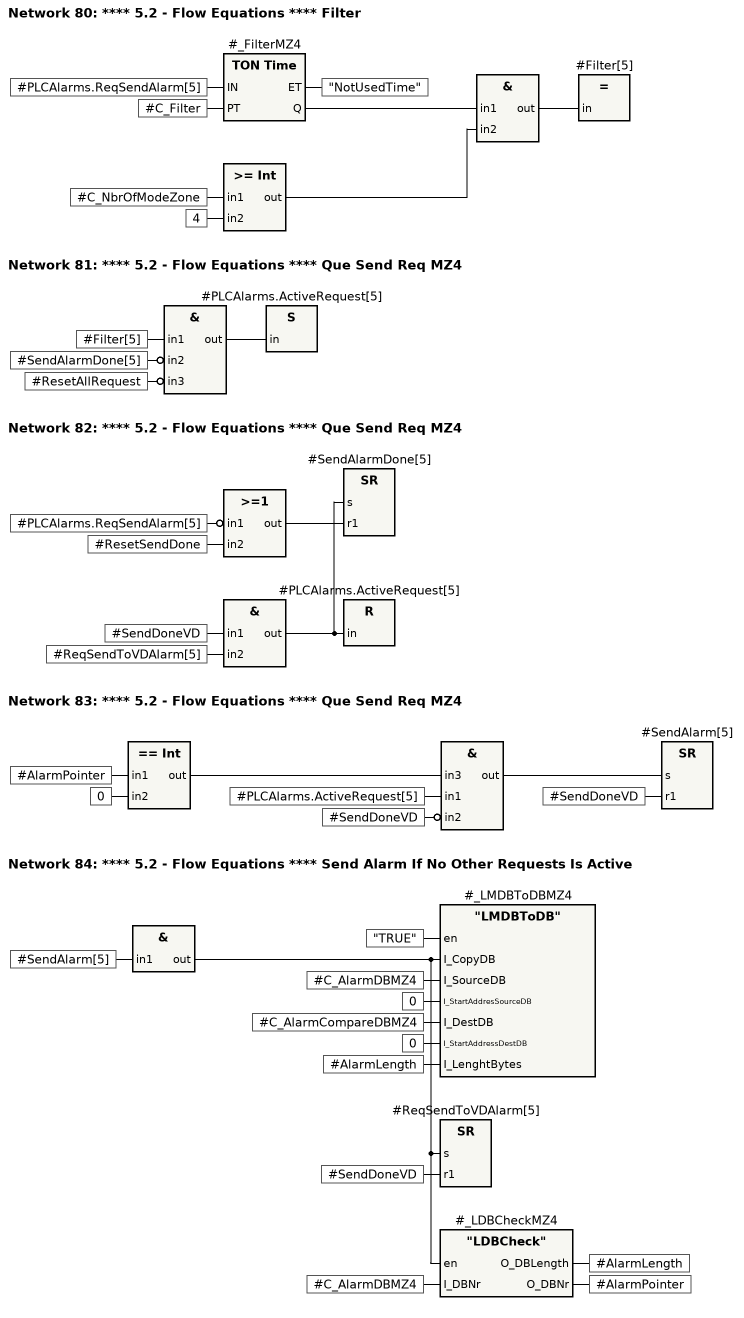
   #_FilterMZ4(IN := #PLCAlarms.ReqSendAlarm[5], PT := #C_Filter, ET => "NotUsedTime");   // TON
   #Filter[5] := #_FilterMZ4.Q AND (#C_NbrOfModeZone >= 4);
END_REGION

REGION Network 81: **** 5.2 - Flow Equations **** Que Send Req MZ4
   // Que Send Req
   IF #Filter[5] AND NOT #SendAlarmDone[5] AND NOT #ResetAllRequest THEN
       #PLCAlarms.ActiveRequest[5] := TRUE;
   END_IF;
END_REGION

REGION Network 82: **** 5.2 - Flow Equations **** Que Send Req MZ4
   // Que Send Req
   #_w1 := #SendDoneVD AND #ReqSendToVDAlarm[5];
   IF #_w1 THEN
       #SendAlarmDone[5] := TRUE;   // SR flip-flop
   END_IF;
   IF NOT #PLCAlarms.ReqSendAlarm[5] OR #ResetSendDone THEN #SendAlarmDone[5] := FALSE; END_IF;
   IF #_w1 THEN #PLCAlarms.ActiveRequest[5] := FALSE; END_IF;
END_REGION

REGION Network 83: **** 5.2 - Flow Equations **** Que Send Req MZ4
   // Que Send Req
   IF (#AlarmPointer = 0) AND #PLCAlarms.ActiveRequest[5] AND NOT #SendDoneVD THEN
       #SendAlarm[5] := TRUE;   // SR flip-flop
   END_IF;
   IF #SendDoneVD THEN #SendAlarm[5] := FALSE; END_IF;
END_REGION

REGION Network 84: **** 5.2 - Flow Equations **** Send Alarm If No Other Requests Is Active
   // Send Alarm If No Other Requests Is Active
   IF #SendAlarm[5] THEN
       #ReqSendToVDAlarm[5] := TRUE;   // SR flip-flop
   END_IF;
   IF #SendDoneVD THEN #ReqSendToVDAlarm[5] := FALSE; END_IF;
   IF #SendAlarm[5] THEN
       #_LDBCheckMZ4(I_DBNr := #C_AlarmDBMZ4, O_DBLength => #AlarmLength, O_DBNr => #AlarmPointer);   // "LDBCheck"
   END_IF;
   IF "TRUE" THEN
       #_LMDBToDBMZ4(I_CopyDB := #SendAlarm[5],   // "LMDBToDB"
                     I_SourceDB := #C_AlarmDBMZ4,
                     I_StartAddresSourceDB := 0,
                     I_DestDB := #C_AlarmCompareDBMZ4,
                     I_StartAddressDestDB := 0,
                     I_LenghtBytes := #AlarmLength);
   END_IF;
END_REGION

REGION Network 85: **** 5.2 - Flow Equations **** Filter
   // Filter
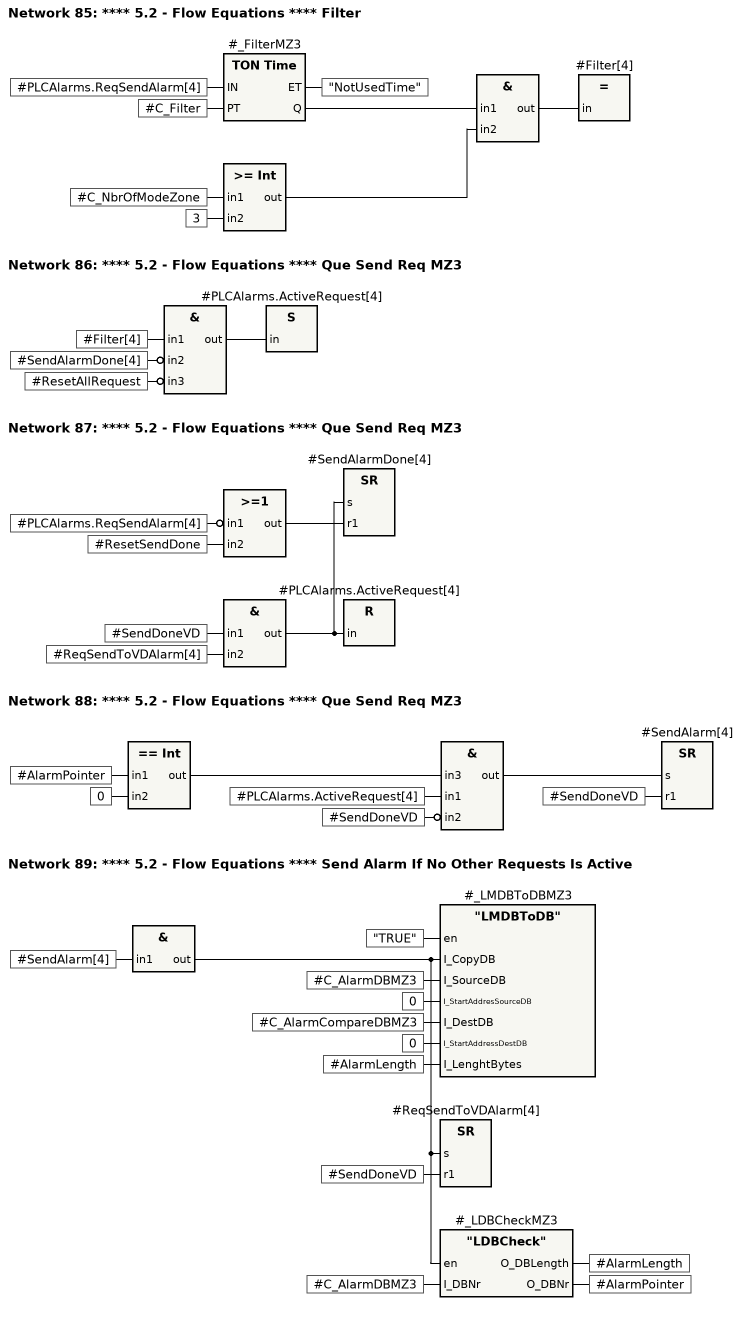
   #_FilterMZ3(IN := #PLCAlarms.ReqSendAlarm[4], PT := #C_Filter, ET => "NotUsedTime");   // TON
   #Filter[4] := #_FilterMZ3.Q AND (#C_NbrOfModeZone >= 3);
END_REGION

REGION Network 86: **** 5.2 - Flow Equations **** Que Send Req MZ3
   // Que Send Req
   IF #Filter[4] AND NOT #SendAlarmDone[4] AND NOT #ResetAllRequest THEN
       #PLCAlarms.ActiveRequest[4] := TRUE;
   END_IF;
END_REGION

REGION Network 87: **** 5.2 - Flow Equations **** Que Send Req MZ3
   // Que Send Req
   #_w1 := #SendDoneVD AND #ReqSendToVDAlarm[4];
   IF #_w1 THEN
       #SendAlarmDone[4] := TRUE;   // SR flip-flop
   END_IF;
   IF NOT #PLCAlarms.ReqSendAlarm[4] OR #ResetSendDone THEN #SendAlarmDone[4] := FALSE; END_IF;
   IF #_w1 THEN #PLCAlarms.ActiveRequest[4] := FALSE; END_IF;
END_REGION

REGION Network 88: **** 5.2 - Flow Equations **** Que Send Req MZ3
   // Que Send Req
   IF (#AlarmPointer = 0) AND #PLCAlarms.ActiveRequest[4] AND NOT #SendDoneVD THEN
       #SendAlarm[4] := TRUE;   // SR flip-flop
   END_IF;
   IF #SendDoneVD THEN #SendAlarm[4] := FALSE; END_IF;
END_REGION

REGION Network 89: **** 5.2 - Flow Equations **** Send Alarm If No Other Requests Is Active
   // Send Alarm If No Other Requests Is Active
   IF #SendAlarm[4] THEN
       #ReqSendToVDAlarm[4] := TRUE;   // SR flip-flop
   END_IF;
   IF #SendDoneVD THEN #ReqSendToVDAlarm[4] := FALSE; END_IF;
   IF #SendAlarm[4] THEN
       #_LDBCheckMZ3(I_DBNr := #C_AlarmDBMZ3, O_DBLength => #AlarmLength, O_DBNr => #AlarmPointer);   // "LDBCheck"
   END_IF;
   IF "TRUE" THEN
       #_LMDBToDBMZ3(I_CopyDB := #SendAlarm[4],   // "LMDBToDB"
                     I_SourceDB := #C_AlarmDBMZ3,
                     I_StartAddresSourceDB := 0,
                     I_DestDB := #C_AlarmCompareDBMZ3,
                     I_StartAddressDestDB := 0,
                     I_LenghtBytes := #AlarmLength);
   END_IF;
END_REGION

REGION Network 90: **** 5.2 - Flow Equations **** Filter
   // Filter
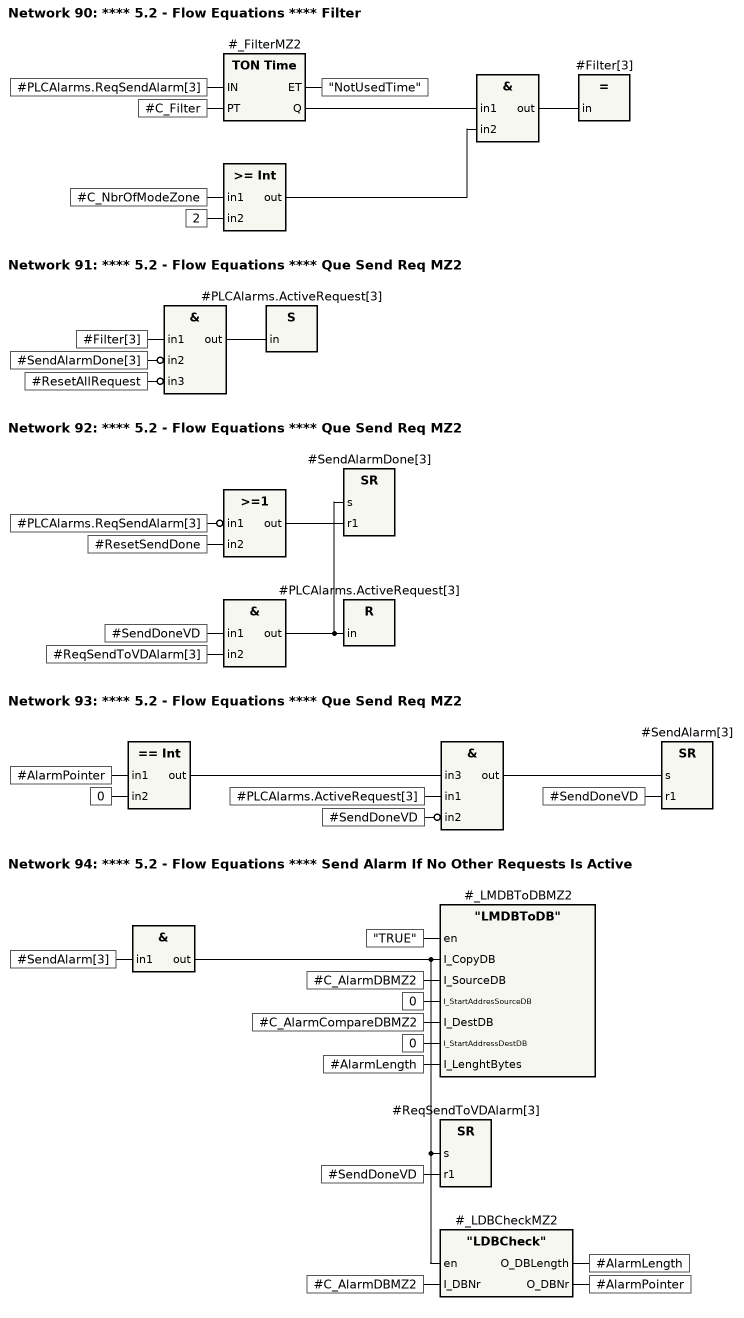
   #_FilterMZ2(IN := #PLCAlarms.ReqSendAlarm[3], PT := #C_Filter, ET => "NotUsedTime");   // TON
   #Filter[3] := #_FilterMZ2.Q AND (#C_NbrOfModeZone >= 2);
END_REGION

REGION Network 91: **** 5.2 - Flow Equations **** Que Send Req MZ2
   // Que Send Req
   IF #Filter[3] AND NOT #SendAlarmDone[3] AND NOT #ResetAllRequest THEN
       #PLCAlarms.ActiveRequest[3] := TRUE;
   END_IF;
END_REGION

REGION Network 92: **** 5.2 - Flow Equations **** Que Send Req MZ2
   // Que Send Req
   #_w1 := #SendDoneVD AND #ReqSendToVDAlarm[3];
   IF #_w1 THEN
       #SendAlarmDone[3] := TRUE;   // SR flip-flop
   END_IF;
   IF NOT #PLCAlarms.ReqSendAlarm[3] OR #ResetSendDone THEN #SendAlarmDone[3] := FALSE; END_IF;
   IF #_w1 THEN #PLCAlarms.ActiveRequest[3] := FALSE; END_IF;
END_REGION

REGION Network 93: **** 5.2 - Flow Equations **** Que Send Req MZ2
   // Que Send Req
   IF (#AlarmPointer = 0) AND #PLCAlarms.ActiveRequest[3] AND NOT #SendDoneVD THEN
       #SendAlarm[3] := TRUE;   // SR flip-flop
   END_IF;
   IF #SendDoneVD THEN #SendAlarm[3] := FALSE; END_IF;
END_REGION

REGION Network 94: **** 5.2 - Flow Equations **** Send Alarm If No Other Requests Is Active
   // Send Alarm If No Other Requests Is Active
   IF #SendAlarm[3] THEN
       #ReqSendToVDAlarm[3] := TRUE;   // SR flip-flop
   END_IF;
   IF #SendDoneVD THEN #ReqSendToVDAlarm[3] := FALSE; END_IF;
   IF #SendAlarm[3] THEN
       #_LDBCheckMZ2(I_DBNr := #C_AlarmDBMZ2, O_DBLength => #AlarmLength, O_DBNr => #AlarmPointer);   // "LDBCheck"
   END_IF;
   IF "TRUE" THEN
       #_LMDBToDBMZ2(I_CopyDB := #SendAlarm[3],   // "LMDBToDB"
                     I_SourceDB := #C_AlarmDBMZ2,
                     I_StartAddresSourceDB := 0,
                     I_DestDB := #C_AlarmCompareDBMZ2,
                     I_StartAddressDestDB := 0,
                     I_LenghtBytes := #AlarmLength);
   END_IF;
END_REGION

REGION Network 95: **** 5.2 - Flow Equations **** Filter
   // Filter
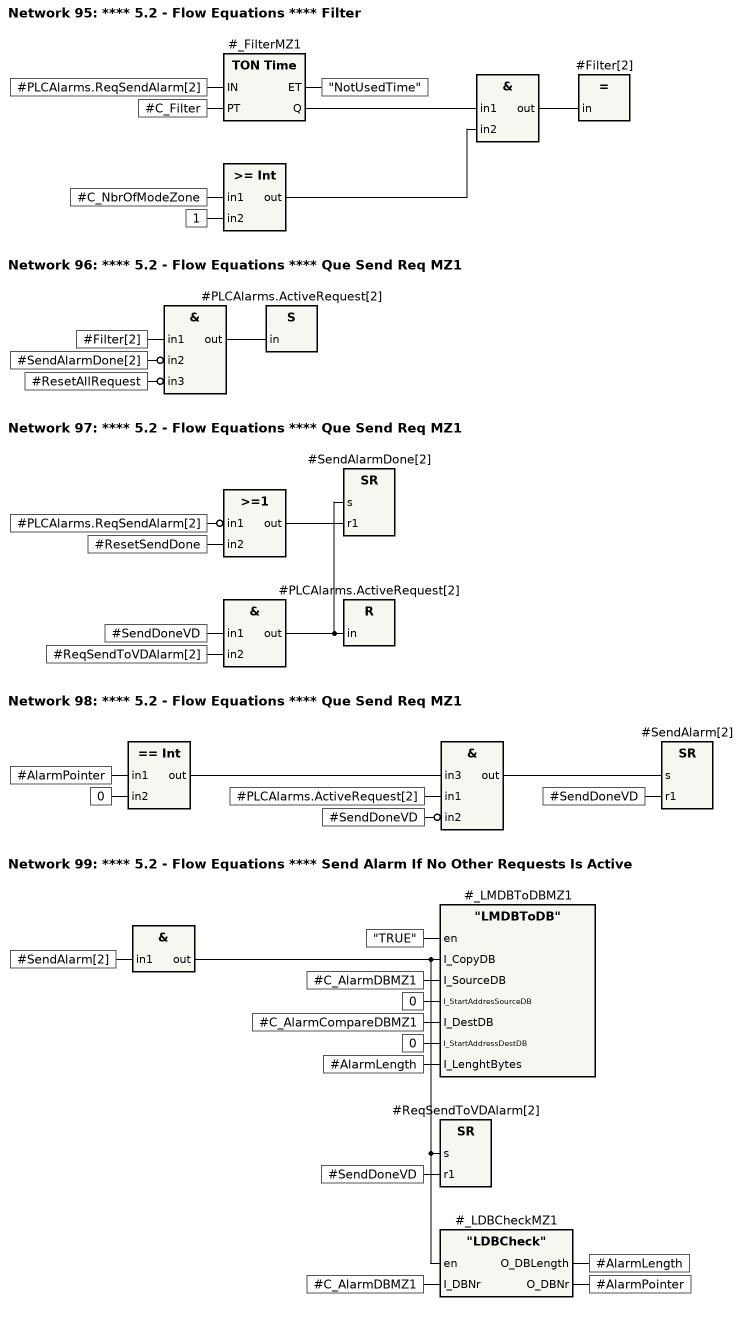
   #_FilterMZ1(IN := #PLCAlarms.ReqSendAlarm[2], PT := #C_Filter, ET => "NotUsedTime");   // TON
   #Filter[2] := #_FilterMZ1.Q AND (#C_NbrOfModeZone >= 1);
END_REGION

REGION Network 96: **** 5.2 - Flow Equations **** Que Send Req MZ1
   // Que Send Req
   IF #Filter[2] AND NOT #SendAlarmDone[2] AND NOT #ResetAllRequest THEN
       #PLCAlarms.ActiveRequest[2] := TRUE;
   END_IF;
END_REGION

REGION Network 97: **** 5.2 - Flow Equations **** Que Send Req MZ1
   // Que Send Req
   #_w1 := #SendDoneVD AND #ReqSendToVDAlarm[2];
   IF #_w1 THEN
       #SendAlarmDone[2] := TRUE;   // SR flip-flop
   END_IF;
   IF NOT #PLCAlarms.ReqSendAlarm[2] OR #ResetSendDone THEN #SendAlarmDone[2] := FALSE; END_IF;
   IF #_w1 THEN #PLCAlarms.ActiveRequest[2] := FALSE; END_IF;
END_REGION

REGION Network 98: **** 5.2 - Flow Equations **** Que Send Req MZ1
   // Que Send Req
   IF (#AlarmPointer = 0) AND #PLCAlarms.ActiveRequest[2] AND NOT #SendDoneVD THEN
       #SendAlarm[2] := TRUE;   // SR flip-flop
   END_IF;
   IF #SendDoneVD THEN #SendAlarm[2] := FALSE; END_IF;
END_REGION

REGION Network 99: **** 5.2 - Flow Equations **** Send Alarm If No Other Requests Is Active
   // Send Alarm If No Other Requests Is Active
   IF #SendAlarm[2] THEN
       #ReqSendToVDAlarm[2] := TRUE;   // SR flip-flop
   END_IF;
   IF #SendDoneVD THEN #ReqSendToVDAlarm[2] := FALSE; END_IF;
   IF #SendAlarm[2] THEN
       #_LDBCheckMZ1(I_DBNr := #C_AlarmDBMZ1, O_DBLength => #AlarmLength, O_DBNr => #AlarmPointer);   // "LDBCheck"
   END_IF;
   IF "TRUE" THEN
       #_LMDBToDBMZ1(I_CopyDB := #SendAlarm[2],   // "LMDBToDB"
                     I_SourceDB := #C_AlarmDBMZ1,
                     I_StartAddresSourceDB := 0,
                     I_DestDB := #C_AlarmCompareDBMZ1,
                     I_StartAddressDestDB := 0,
                     I_LenghtBytes := #AlarmLength);
   END_IF;
END_REGION

REGION Network 100: **** 5.2 - Flow Equations **** Filter
   // Filter
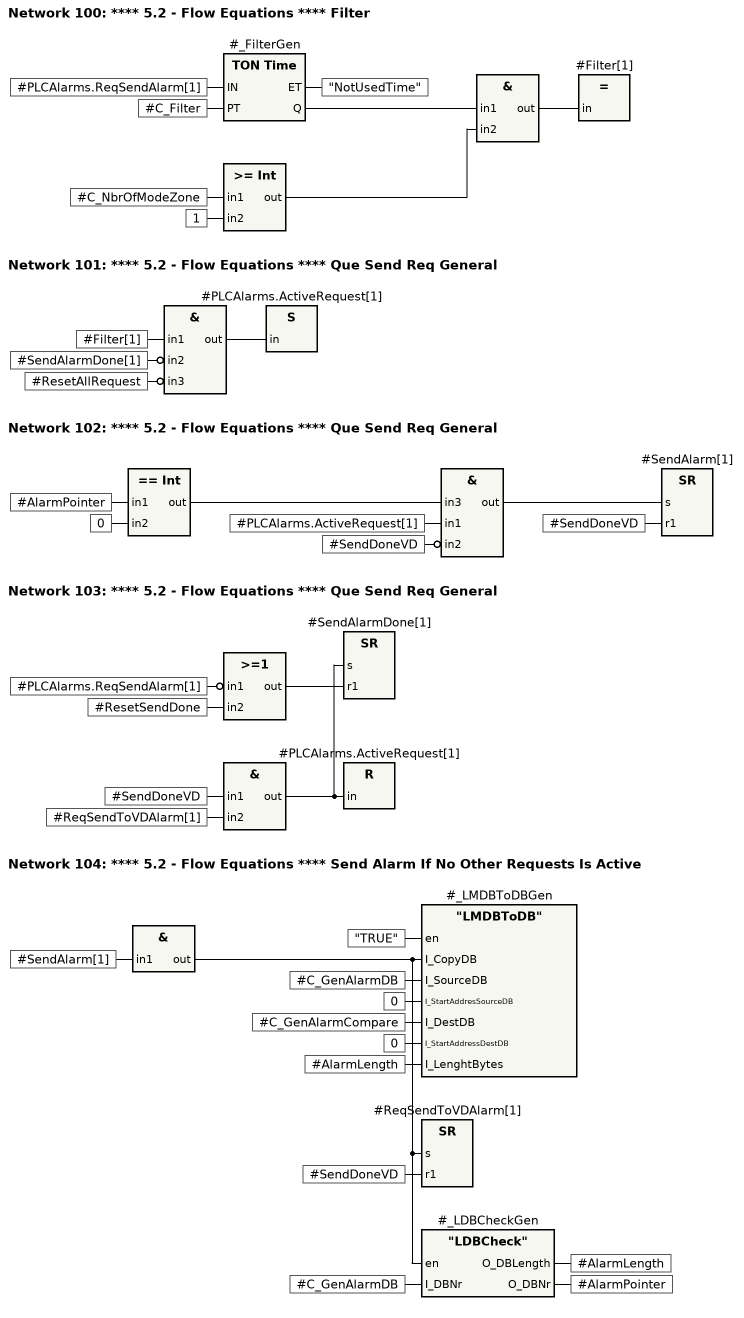
   #_FilterGen(IN := #PLCAlarms.ReqSendAlarm[1], PT := #C_Filter, ET => "NotUsedTime");   // TON
   #Filter[1] := #_FilterGen.Q AND (#C_NbrOfModeZone >= 1);
END_REGION

REGION Network 101: **** 5.2 - Flow Equations **** Que Send Req General
   // Que Send Req
   IF #Filter[1] AND NOT #SendAlarmDone[1] AND NOT #ResetAllRequest THEN
       #PLCAlarms.ActiveRequest[1] := TRUE;
   END_IF;
END_REGION

REGION Network 102: **** 5.2 - Flow Equations **** Que Send Req General
   // Que Send Req
   IF (#AlarmPointer = 0) AND #PLCAlarms.ActiveRequest[1] AND NOT #SendDoneVD THEN
       #SendAlarm[1] := TRUE;   // SR flip-flop
   END_IF;
   IF #SendDoneVD THEN #SendAlarm[1] := FALSE; END_IF;
END_REGION

REGION Network 103: **** 5.2 - Flow Equations **** Que Send Req General
   // Que Send Req
   #_w1 := #SendDoneVD AND #ReqSendToVDAlarm[1];
   IF #_w1 THEN
       #SendAlarmDone[1] := TRUE;   // SR flip-flop
   END_IF;
   IF NOT #PLCAlarms.ReqSendAlarm[1] OR #ResetSendDone THEN #SendAlarmDone[1] := FALSE; END_IF;
   IF #_w1 THEN #PLCAlarms.ActiveRequest[1] := FALSE; END_IF;
END_REGION

REGION Network 104: **** 5.2 - Flow Equations **** Send Alarm If No Other Requests Is Active
   // Send Alarm If No Other Requests Is Active
   IF #SendAlarm[1] THEN
       #ReqSendToVDAlarm[1] := TRUE;   // SR flip-flop
   END_IF;
   IF #SendDoneVD THEN #ReqSendToVDAlarm[1] := FALSE; END_IF;
   IF #SendAlarm[1] THEN
       #_LDBCheckGen(I_DBNr := #C_GenAlarmDB, O_DBLength => #AlarmLength, O_DBNr => #AlarmPointer);   // "LDBCheck"
   END_IF;
   IF "TRUE" THEN
       #_LMDBToDBGen(I_CopyDB := #SendAlarm[1],   // "LMDBToDB"
                     I_SourceDB := #C_GenAlarmDB,
                     I_StartAddresSourceDB := 0,
                     I_DestDB := #C_GenAlarmCompare,
                     I_StartAddressDestDB := 0,
                     I_LenghtBytes := #AlarmLength);
   END_IF;
END_REGION
END_FUNCTION_BLOCK
